KUKA KRL program: MyProgram_265().src

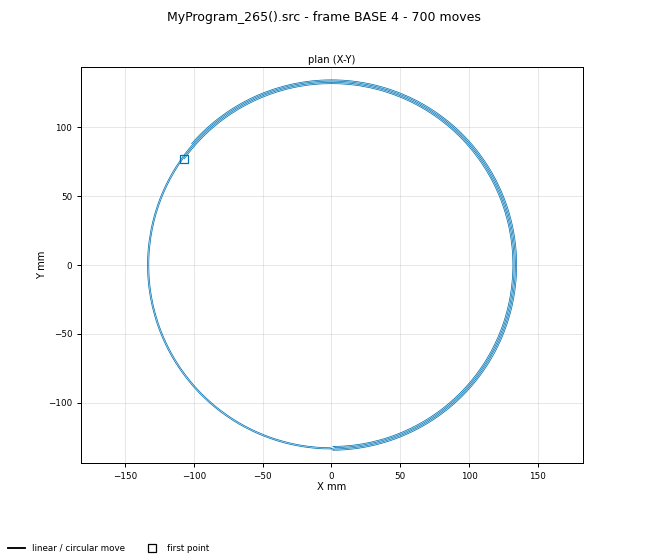
[picture p0: tool path of MyProgram_265().src in frame BASE 4, 700 of 700 moves have a stored position in this frame; points joined in program order, loops and branches not executed]
&ACCESS RVP
&REL 1
&PARAM TEMPLATE = C:\KRC\Roboter\Template\vorgabe
&PARAM EDITMASK = *
DEF MyProgram_265()
; ---- Setting reference (Base) ----
$BASE = BASE_DATA[4]

; --------------------------
; ---- Setting tool (TCP) ----
$TOOL = TOOL_DATA[3]
; --------------------------

$VEL.CP = VEL_APROX_PRINT
Startdeposition()
$VEL.CP = VEL_PRINT
LIN {X -106.8774,Y 77.2137,Z 169,A 144.3392,B 9.9671,C 0.0916,E1 9.8386,E2 306.7155} C_DIS
LIN {X -104.49,Y 80.4156,Z 169,A 142.5484,B 9.9671,C 0.0885,E1 9.8417,E2 308.5109} C_DIS
LIN {X -101.9162,Y 83.6531,Z 169,A 140.5928,B 9.9671,C 0.0871,E1 9.8451,E2 310.483} C_DIS
LIN {X -98.7876,Y 87.3252,Z 169,A 138.4779,B 9.9672,C 0.0828,E1 9.849,E2 312.5979} C_DIS
LIN {X -95.5133,Y 90.8953,Z 169,A 136.3519,B 9.9672,C 0.0786,E1 9.853,E2 314.724} C_DIS
LIN {X -92.6386,Y 93.824,Z 169,A 134.5368,B 9.9672,C 0.0754,E1 9.8566,E2 316.5411} C_DIS
LIN {X -89.1298,Y 97.1626,Z 169,A 132.4198,B 9.9672,C 0.0714,E1 9.8609,E2 318.6574} C_DIS
LIN {X -85.5317,Y 100.3446,Z 169,A 130.3464,B 9.9673,C 0.067,E1 9.8653,E2 320.7271} C_DIS
LIN {X -82.2873,Y 103.022,Z 169,A 128.4814,B 9.9673,C 0.0643,E1 9.8694,E2 322.5946} C_DIS
LIN {X -78.5317,Y 105.9128,Z 169,A 126.5407,B 9.9673,C 0.0584,E1 9.8736,E2 324.5197} C_DIS
LIN {X -75.9379,Y 107.7874,Z 169,A 125.1409,B 9.9673,C 0.0562,E1 9.8768,E2 325.9191} C_DIS
LIN {X -73.2593,Y 109.6255,Z 169,A 123.7103,B 9.9674,C 0.0542,E1 9.8801,E2 327.3506} C_DIS
LIN {X -70.5616,Y 111.3813,Z 169,A 122.3083,B 9.9674,C 0.052,E1 9.8834,E2 328.7518} C_DIS
LIN {X -67.8103,Y 113.0777,Z 169,A 120.8832,B 9.9674,C 0.0502,E1 9.8868,E2 330.1781} C_DIS
LIN {X -64.9859,Y 114.7243,Z 169,A 119.5244,B 9.9674,C 0.0469,E1 9.8901,E2 331.5284} C_DIS
LIN {X -62.1565,Y 116.2813,Z 169,A 118.0193,B 9.9674,C 0.0469,E1 9.8938,E2 333.0441} C_DIS
LIN {X -59.3244,Y 117.75,Z 169,A 116.6411,B 9.9674,C 0.0448,E1 9.8972,E2 334.4201} C_DIS
LIN {X -56.4217,Y 119.1678,Z 169,A 115.2277,B 9.9674,C 0.0431,E1 9.9008,E2 335.8334} C_DIS
LIN {X -53.4693,Y 120.5212,Z 169,A 113.8101,B 9.9674,C 0.0415,E1 9.9044,E2 337.2506} C_DIS
LIN {X -50.4743,Y 121.8058,Z 169,A 112.3819,B 9.9674,C 0.0401,E1 9.9081,E2 338.6791} C_DIS
LIN {X -47.4755,Y 123.0055,Z 169,A 110.9758,B 9.9674,C 0.0386,E1 9.9117,E2 340.0844} C_DIS
LIN {X -44.4123,Y 124.1444,Z 169,A 109.5673,B 9.9674,C 0.0369,E1 9.9154,E2 341.4904} C_DIS
LIN {X -41.359,Y 125.1947,Z 169,A 108.139,B 9.9674,C 0.036,E1 9.9192,E2 342.9206} C_DIS
LIN {X -38.2477,Y 126.1802,Z 169,A 106.716,B 9.9674,C 0.0348,E1 9.923,E2 344.3431} C_DIS
LIN {X -35.201,Y 127.0638,Z 169,A 105.3278,B 9.9674,C 0.0339,E1 9.9267,E2 345.7315} C_DIS
LIN {X -32.095,Y 127.8837,Z 169,A 103.9426,B 9.9674,C 0.0326,E1 9.9305,E2 347.1145} C_DIS
LIN {X -28.9319,Y 128.6366,Z 169,A 102.5542,B 9.9675,C 0.0311,E1 9.9342,E2 348.4991} C_DIS
LIN {X -25.7137,Y 129.3189,Z 169,A 101.0837,B 9.9675,C 0.0311,E1 9.9383,E2 349.9734} C_DIS
LIN {X -22.5381,Y 129.9106,Z 169,A 99.6804,B 9.9675,C 0.0303,E1 9.9421,E2 351.3759} C_DIS
LIN {X -19.3867,Y 130.4184,Z 169,A 98.2497,B 9.9675,C 0.0304,E1 9.9461,E2 352.8108} C_DIS
LIN {X -16.181,Y 130.854,Z 169,A 96.9617,B 9.9675,C 0.0275,E1 9.9496,E2 354.0843} C_DIS
LIN {X -12.9527,Y 131.2122,Z 169,A 95.4376,B 9.9675,C 0.0293,E1 9.9539,E2 355.6206} C_DIS
LIN {X -10.1839,Y 131.4569,Z 169,A 94.1244,B 9.9675,C 0.0311,E1 9.9576,E2 356.9454} C_DIS
LIN {X -6.5072,Y 131.6889,Z 169,A 92.6483,B 9.9675,C 0.0282,E1 9.9616,E2 358.4062} C_DIS
LIN {X -3.2367,Y 131.8105,Z 169,A 91.2707,B 9.9675,C 0.0272,E1 9.9655,E2 359.778} C_DIS
LIN {X -0.026,Y 131.8515,Z 169,A 89.7952,B 9.9675,C 0.0287,E1 9.9696,E2 361.2622} C_DIS
LIN {X 3.2431,Y 131.8103,Z 169,A 88.5531,B 9.9675,C 0.0251,E1 9.973,E2 362.4828} C_DIS
LIN {X 6.4726,Y 131.6906,Z 169,A 86.9955,B 9.9675,C 0.0283,E1 9.9774,E2 364.0576} C_DIS
LIN {X 9.6971,Y 131.4924,Z 169,A 85.5991,B 9.9675,C 0.0284,E1 9.9813,E2 365.4526} C_DIS
LIN {X 12.9671,Y 131.2108,Z 169,A 84.0255,B 9.9675,C 0.0318,E1 9.9857,E2 367.0428} C_DIS
LIN {X 17.2713,Y 130.7134,Z 169,A 82.2451,B 9.9675,C 0.0303,E1 9.9906,E2 368.8107} C_DIS
LIN {X 20.945,Y 130.1773,Z 169,A 80.6692,B 9.9675,C 0.0302,E1 9.995,E2 370.3819} C_DIS
LIN {X 24.0929,Y 129.6311,Z 169,A 79.2883,B 9.9675,C 0.0307,E1 9.9987,E2 371.7615} C_DIS
LIN {X 27.2612,Y 129.0015,Z 169,A 77.8766,B 9.9675,C 0.0316,E1 10.0026,E2 373.1737} C_DIS
LIN {X 30.4672,Y 128.2816,Z 169,A 76.4611,B 9.9675,C 0.0322,E1 10.0065,E2 374.5874} C_DIS
LIN {X 33.0736,Y 127.6354,Z 169,A 75.1852,B 9.9675,C 0.0353,E1 10.0099,E2 375.8757} C_DIS
LIN {X 36.7115,Y 126.6357,Z 169,A 73.6812,B 9.9675,C 0.0337,E1 10.0139,E2 377.3637} C_DIS
LIN {X 39.7849,Y 125.7039,Z 169,A 72.2874,B 9.9675,C 0.0348,E1 10.0177,E2 378.7571} C_DIS
LIN {X 42.8518,Y 124.6918,Z 169,A 70.9049,B 9.9675,C 0.0356,E1 10.0213,E2 380.1369} C_DIS
LIN {X 45.9047,Y 123.6004,Z 169,A 69.4777,B 9.9675,C 0.0374,E1 10.0251,E2 381.5662} C_DIS
LIN {X 48.9596,Y 122.4225,Z 169,A 68.0862,B 9.9675,C 0.0382,E1 10.0287,E2 382.9539} C_DIS
LIN {X 51.9473,Y 121.185,Z 169,A 66.679,B 9.9675,C 0.0398,E1 10.0323,E2 384.3612} C_DIS
LIN {X 54.905,Y 119.8742,Z 169,A 65.3074,B 9.9675,C 0.0407,E1 10.0358,E2 385.7289} C_DIS
LIN {X 57.3093,Y 118.7437,Z 169,A 64.0084,B 9.9675,C 0.0452,E1 10.0391,E2 387.0447} C_DIS
LIN {X 60.2841,Y 117.2615,Z 169,A 62.6301,B 9.9675,C 0.0456,E1 10.0425,E2 388.4154} C_DIS
LIN {X 63.5459,Y 115.5281,Z 169,A 61.1059,B 9.9675,C 0.046,E1 10.0462,E2 389.9303} C_DIS
LIN {X 66.3562,Y 113.9371,Z 169,A 59.7046,B 9.9675,C 0.048,E1 10.0496,E2 391.3314} C_DIS
LIN {X 69.1671,Y 112.2527,Z 169,A 58.2922,B 9.9675,C 0.0498,E1 10.053,E2 392.7426} C_DIS
LIN {X 71.9319,Y 110.5012,Z 169,A 56.8911,B 9.9675,C 0.0516,E1 10.0563,E2 394.1415} C_DIS
LIN {X 74.5745,Y 108.7351,Z 169,A 55.5407,B 9.9675,C 0.0531,E1 10.0594,E2 395.4885} C_DIS
LIN {X 77.241,Y 106.8575,Z 169,A 54.1443,B 9.9675,C 0.055,E1 10.0626,E2 396.8827} C_DIS
LIN {X 79.8287,Y 104.9389,Z 169,A 52.7306,B 9.9674,C 0.0577,E1 10.0657,E2 398.2984} C_DIS
LIN {X 82.4043,Y 102.9288,Z 169,A 51.1566,B 9.9674,C 0.0636,E1 10.0692,E2 399.8907} C_DIS
LIN {X 85.5078,Y 100.3649,Z 169,A 49.427,B 9.9674,C 0.0664,E1 10.0729,E2 401.6185} C_DIS
LIN {X 88.551,Y 97.6904,Z 169,A 47.6868,B 9.9674,C 0.0693,E1 10.0765,E2 403.3568} C_DIS
LIN {X 92.0675,Y 94.3843,Z 169,A 45.7593,B 9.9674,C 0.0697,E1 10.0804,E2 405.2652} C_DIS
LIN {X 94.9298,Y 91.5046,Z 169,A 43.8603,B 9.9673,C 0.0763,E1 10.0841,E2 407.1806} C_DIS
LIN {X 97.7032,Y 88.5369,Z 169,A 42.1172,B 9.9673,C 0.0796,E1 10.0874,E2 408.9218} C_DIS
LIN {X 100.3808,Y 85.4891,Z 169,A 40.3789,B 9.9673,C 0.0828,E1 10.0906,E2 410.658} C_DIS
LIN {X 102.9666,Y 82.3569,Z 169,A 38.639,B 9.9672,C 0.0862,E1 10.0936,E2 412.3958} C_DIS
LIN {X 105.8792,Y 78.5769,Z 169,A 36.7305,B 9.9672,C 0.0872,E1 10.0968,E2 414.2859} C_DIS
LIN {X 107.3485,Y 76.5572,Z 169,A 35.5161,B 9.9672,C 0.0927,E1 10.0988,E2 415.516} C_DIS
LIN {X 109.6294,Y 73.2536,Z 169,A 33.9386,B 9.9672,C 0.093,E1 10.1013,E2 417.0748} C_DIS
LIN {X 111.3712,Y 70.5777,Z 169,A 32.5709,B 9.9671,C 0.0959,E1 10.1033,E2 418.441} C_DIS
LIN {X 113.0732,Y 67.8178,Z 169,A 31.1149,B 9.9671,C 0.1005,E1 10.1055,E2 419.9033} C_DIS
LIN {X 114.7841,Y 64.8799,Z 169,A 29.7352,B 9.9671,C 0.1019,E1 10.1074,E2 421.2725} C_DIS
LIN {X 116.2924,Y 62.1357,Z 169,A 28.3549,B 9.967,C 0.1058,E1 10.1092,E2 422.6559} C_DIS
LIN {X 117.7557,Y 59.3133,Z 169,A 27.0047,B 9.967,C 0.1087,E1 10.1109,E2 424.0033} C_DIS
LIN {X 119.1743,Y 56.4081,Z 169,A 25.62,B 9.967,C 0.1118,E1 10.1126,E2 425.3865} C_DIS
LIN {X 120.5203,Y 53.4713,Z 169,A 24.2359,B 9.9669,C 0.1151,E1 10.1142,E2 426.7693} C_DIS
LIN {X 121.7955,Y 50.499,Z 169,A 22.8442,B 9.9669,C 0.1185,E1 10.1157,E2 428.1603} C_DIS
LIN {X 123.0031,Y 47.4818,Z 169,A 21.4588,B 9.9669,C 0.1217,E1 10.1171,E2 429.5436} C_DIS
LIN {X 124.1429,Y 44.4166,Z 169,A 20.0581,B 9.9668,C 0.1251,E1 10.1184,E2 430.9429} C_DIS
LIN {X 125.0907,Y 41.6715,Z 169,A 18.7574,B 9.9668,C 0.1294,E1 10.1196,E2 432.2491} C_DIS
LIN {X 126.1752,Y 38.2641,Z 169,A 17.2961,B 9.9667,C 0.1316,E1 10.1208,E2 433.7007} C_DIS
LIN {X 127.0596,Y 35.2158,Z 169,A 16.006,B 9.9667,C 0.1333,E1 10.1218,E2 434.9813} C_DIS
LIN {X 127.8876,Y 32.0798,Z 169,A 14.5795,B 9.9667,C 0.1377,E1 10.1228,E2 436.4111} C_DIS
LIN {X 128.5443,Y 29.3357,Z 169,A 13.2661,B 9.9665,C 0.1432,E1 10.1236,E2 437.7358} C_DIS
LIN {X 129.3167,Y 25.7247,Z 169,A 11.7507,B 9.9665,C 0.1457,E1 10.1245,E2 439.242} C_DIS
LIN {X 129.9091,Y 22.5464,Z 169,A 10.3707,B 9.9665,C 0.1491,E1 10.1252,E2 440.6204} C_DIS
LIN {X 130.4172,Y 19.395,Z 169,A 8.9639,B 9.9664,C 0.1536,E1 10.1258,E2 442.0308} C_DIS
LIN {X 130.8537,Y 16.1835,Z 169,A 7.6069,B 9.9664,C 0.1564,E1 10.1263,E2 443.3828} C_DIS
LIN {X 131.2111,Y 12.9638,Z 169,A 6.1987,B 9.9663,C 0.1605,E1 10.1267,E2 444.7924} C_DIS
LIN {X 131.4627,Y 10.1046,Z 169,A 4.8935,B 9.9662,C 0.1655,E1 10.127,E2 446.1056} C_DIS
LIN {X 131.6884,Y 6.5173,Z 169,A 3.4541,B 9.9662,C 0.1671,E1 10.1272,E2 447.5319} C_DIS
LIN {X 131.8107,Y 3.2292,Z 169,A 2.061,B 9.9662,C 0.1704,E1 10.1273,E2 448.9221} C_DIS
LIN {X 131.8522,Y 0.2318,Z 169,A 0.6856,B 9.966,C 0.176,E1 10.1273,E2 450.3075} C_DIS
LIN {X 131.8106,Y -3.2343,Z 169,A -0.7295,B 9.966,C 0.1782,E1 10.1273,E2 451.713} C_DIS
LIN {X 131.691,Y -6.4646,Z 169,A -2.015,B 9.966,C 0.1795,E1 10.1271,E2 452.9857} C_DIS
LIN {X 131.4921,Y -9.7022,Z 169,A -3.4963,B 9.9658,C 0.1853,E1 10.1269,E2 454.477} C_DIS
LIN {X 131.2186,Y -12.8854,Z 169,A -4.8644,B 9.9658,C 0.1889,E1 10.1265,E2 455.8441} C_DIS
LIN {X 130.859,Y -16.1387,Z 169,A -6.2578,B 9.9658,C 0.1923,E1 10.1261,E2 457.2355} C_DIS
LIN {X 130.431,Y -19.2984,Z 169,A -7.6232,B 9.9656,C 0.1959,E1 10.1255,E2 458.6} C_DIS
LIN {X 129.9116,Y -22.5325,Z 169,A -8.9978,B 9.9656,C 0.1988,E1 10.1249,E2 459.9701} C_DIS
LIN {X 129.326,Y -25.6791,Z 169,A -10.4159,B 9.9655,C 0.2035,E1 10.1242,E2 461.393} C_DIS
LIN {X 128.6466,Y -28.888,Z 169,A -11.816,B 9.9655,C 0.207,E1 10.1233,E2 462.7915} C_DIS
LIN {X 127.8992,Y -32.0341,Z 169,A -13.2076,B 9.9653,C 0.2107,E1 10.1224,E2 464.183} C_DIS
LIN {X 127.0798,Y -35.1435,Z 169,A -14.5851,B 9.9653,C 0.2142,E1 10.1214,E2 465.5596} C_DIS
LIN {X 126.1828,Y -38.2391,Z 169,A -16.0454,B 9.9652,C 0.2195,E1 10.1202,E2 467.0286} C_DIS
LIN {X 124.9065,Y -42.2245,Z 169,A -17.8958,B 9.965,C 0.2254,E1 10.1186,E2 468.8848} C_DIS
LIN {X 123.6012,Y -45.9026,Z 169,A -19.4299,B 9.965,C 0.2263,E1 10.1172,E2 470.4013} C_DIS
LIN {X 122.4235,Y -48.9571,Z 169,A -20.8082,B 9.965,C 0.2292,E1 10.1158,E2 471.7758} C_DIS
LIN {X 121.1855,Y -51.9463,Z 169,A -22.2141,B 9.9649,C 0.233,E1 10.1142,E2 473.1832} C_DIS
LIN {X 119.8648,Y -54.9253,Z 169,A -23.5996,B 9.9648,C 0.2361,E1 10.1127,E2 474.5666} C_DIS
LIN {X 118.4854,Y -57.8418,Z 169,A -24.9809,B 9.9648,C 0.2394,E1 10.111,E2 475.9469} C_DIS
LIN {X 117.0349,Y -60.7239,Z 169,A -26.3094,B 9.9647,C 0.2414,E1 10.1093,E2 477.2681} C_DIS
LIN {X 115.5353,Y -63.5329,Z 169,A -27.7352,B 9.9645,C 0.246,E1 10.1074,E2 478.7005} C_DIS
LIN {X 113.9475,Y -66.3382,Z 169,A -29.1224,B 9.9645,C 0.2493,E1 10.1055,E2 480.0876} C_DIS
LIN {X 112.2709,Y -69.1374,Z 169,A -30.5256,B 9.9644,C 0.2525,E1 10.1034,E2 481.4906} C_DIS
LIN {X 110.2507,Y -72.3153,Z 169,A -32.2569,B 9.9642,C 0.2589,E1 10.1008,E2 483.2351} C_DIS
LIN {X 107.7951,Y -75.927,Z 169,A -34.0046,B 9.9642,C 0.26,E1 10.0981,E2 484.9667} C_DIS
LIN {X 105.9051,Y -78.5421,Z 169,A -35.386,B 9.9642,C 0.263,E1 10.0958,E2 486.3471} C_DIS
LIN {X 104.4254,Y -80.4992,Z 169,A -36.5931,B 9.964,C 0.2688,E1 10.0937,E2 487.5724} C_DIS
LIN {X 101.8901,Y -83.6851,Z 169,A -38.3507,B 9.9639,C 0.2726,E1 10.0906,E2 489.3304} C_DIS
LIN {X 98.7684,Y -87.3469,Z 169,A -40.4118,B 9.9637,C 0.2767,E1 10.0868,E2 491.3901} C_DIS
LIN {X 95.5049,Y -90.9041,Z 169,A -42.4828,B 9.9637,C 0.2807,E1 10.0829,E2 493.4601} C_DIS
LIN {X 92.6078,Y -93.8543,Z 169,A -44.2682,B 9.9635,C 0.2843,E1 10.0794,E2 495.246} C_DIS
LIN {X 89.1247,Y -97.1673,Z 169,A -46.3322,B 9.9635,C 0.2881,E1 10.0752,E2 497.309} C_DIS
LIN {X 85.5204,Y -100.3542,Z 169,A -48.3987,B 9.9633,C 0.2917,E1 10.0708,E2 499.3747} C_DIS
LIN {X 82.358,Y -102.9657,Z 169,A -50.1566,B 9.9633,C 0.2946,E1 10.067,E2 501.1314} C_DIS
LIN {X 78.5751,Y -105.8805,Z 169,A -52.0711,B 9.9633,C 0.2948,E1 10.0628,E2 503.0285} C_DIS
LIN {X 75.9621,Y -107.7703,Z 169,A -53.4748,B 9.9632,C 0.2974,E1 10.0596,E2 504.4338} C_DIS
LIN {X 72.5727,Y -110.0813,Z 169,A -55.2404,B 9.9631,C 0.3001,E1 10.0555,E2 506.199} C_DIS
LIN {X 69.1643,Y -112.2544,Z 169,A -56.9607,B 9.9631,C 0.3022,E1 10.0514,E2 507.9167} C_DIS
LIN {X 66.3665,Y -113.9311,Z 169,A -58.3647,B 9.963,C 0.3041,E1 10.0481,E2 509.3203} C_DIS
LIN {X 63.5661,Y -115.5169,Z 169,A -59.7625,B 9.9629,C 0.3062,E1 10.0446,E2 510.7193} C_DIS
LIN {X 60.7608,Y -117.0155,Z 169,A -61.1372,B 9.9629,C 0.3081,E1 10.0412,E2 512.0942} C_DIS
LIN {X 57.8826,Y -118.4652,Z 169,A -62.5279,B 9.9628,C 0.3099,E1 10.0378,E2 513.485} C_DIS
LIN {X 54.9401,Y -119.858,Z 169,A -63.9294,B 9.9628,C 0.3115,E1 10.0342,E2 514.8861} C_DIS
LIN {X 51.9832,Y -121.1695,Z 169,A -65.3247,B 9.9627,C 0.313,E1 10.0306,E2 516.2812} C_DIS
LIN {X 48.8175,Y -122.4797,Z 169,A -66.7966,B 9.9627,C 0.3145,E1 10.0268,E2 517.7524} C_DIS
LIN {X 45.9072,Y -123.5995,Z 169,A -68.1518,B 9.9626,C 0.316,E1 10.0233,E2 519.1086} C_DIS
LIN {X 42.8223,Y -124.702,Z 169,A -69.7168,B 9.9624,C 0.3207,E1 10.0191,E2 520.6918} C_DIS
LIN {X 38.8604,Y -125.9927,Z 169,A -71.4795,B 9.9624,C 0.3214,E1 10.0144,E2 522.4501} C_DIS
LIN {X 35.2363,Y -127.0539,Z 169,A -73.0067,B 9.9624,C 0.3205,E1 10.0104,E2 523.9646} C_DIS
LIN {X 32.0725,Y -127.8894,Z 169,A -74.412,B 9.9624,C 0.3213,E1 10.0066,E2 525.369} C_DIS
LIN {X 28.9296,Y -128.6371,Z 169,A -75.8087,B 9.9624,C 0.3223,E1 10.0028,E2 526.7658} C_DIS
LIN {X 25.7271,Y -129.3162,Z 169,A -77.2229,B 9.9624,C 0.3231,E1 9.9989,E2 528.18} C_DIS
LIN {X 22.5399,Y -129.9103,Z 169,A -78.6228,B 9.9624,C 0.3238,E1 9.9951,E2 529.5796} C_DIS
LIN {X 19.3793,Y -130.4195,Z 169,A -80.0488,B 9.9623,C 0.3254,E1 9.9911,E2 531.0108} C_DIS
LIN {X 16.1804,Y -130.854,Z 169,A -81.434,B 9.9623,C 0.3257,E1 9.9873,E2 532.3946} C_DIS
LIN {X 12.9655,Y -131.2109,Z 169,A -82.8418,B 9.9623,C 0.3263,E1 9.9834,E2 533.8035} C_DIS
LIN {X 9.7296,Y -131.4901,Z 169,A -84.235,B 9.9623,C 0.3264,E1 9.9795,E2 535.1952} C_DIS
LIN {X 6.5046,Y -131.689,Z 169,A -85.6292,B 9.9623,C 0.3266,E1 9.9756,E2 536.589} C_DIS
LIN {X 3.2349,Y -131.8106,Z 169,A -87.0343,B 9.9623,C 0.3266,E1 9.9717,E2 537.9928} C_DIS
LIN {X 0.956,Y -131.8451,Z 169,A -87.7495,B 9.9624,C 0.321,E1 9.9698,E2 538.6752} C_DIS
Enddeposition()
LIN {X 0.956,Y -131.8451,Z 169,A -87.7495,B 9.9624,C 0.321,E1 9.9698,E2 538.6752} C_DIS
Startdeposition()
$VEL.CP = VEL_PRINT
LIN {X 3.133,Y -132.7261,Z 169,A -86.3062,B 9.9633,C 0.3159,E1 9.9747,E2 537.2036} C_DIS
LIN {X 6.6755,Y -132.5939,Z 169,A -84.9357,B 9.9633,C 0.319,E1 9.9784,E2 535.852} C_DIS
LIN {X 10.3215,Y -132.3616,Z 169,A -83.3705,B 9.9633,C 0.3187,E1 9.9828,E2 534.2874} C_DIS
LIN {X 13.2936,Y -132.096,Z 169,A -81.9074,B 9.9633,C 0.3144,E1 9.9869,E2 532.802} C_DIS
LIN {X 17.2969,Y -131.6302,Z 169,A -80.3789,B 9.9633,C 0.3181,E1 9.9911,E2 531.2983} C_DIS
LIN {X 20.4371,Y -131.1793,Z 169,A -78.9281,B 9.9633,C 0.3156,E1 9.9951,E2 529.8366} C_DIS
LIN {X 24.5903,Y -130.4649,Z 169,A -77.0814,B 9.9634,C 0.3138,E1 10.0002,E2 527.9854} C_DIS
LIN {X 27.6052,Y -129.8606,Z 169,A -75.7814,B 9.9634,C 0.3134,E1 10.0037,E2 526.6878} C_DIS
LIN {X 30.6136,Y -129.1848,Z 169,A -74.6207,B 9.9634,C 0.3162,E1 10.0068,E2 525.5472} C_DIS
LIN {X 33.4173,Y -128.4894,Z 169,A -73.2702,B 9.9634,C 0.3128,E1 10.0105,E2 524.183} C_DIS
LIN {X 39.0819,Y -126.879,Z 169,A -70.7402,B 9.9635,C 0.3107,E1 10.0173,E2 521.6525} C_DIS
LIN {X 44.8545,Y -124.9548,Z 169,A -68.0494,B 9.9636,C 0.3065,E1 10.0245,E2 518.9518} C_DIS
LIN {X 50.4355,Y -122.8107,Z 169,A -65.5025,B 9.9637,C 0.3042,E1 10.0311,E2 516.4071} C_DIS
LIN {X 53.6522,Y -121.4388,Z 169,A -64.1366,B 9.9637,C 0.3055,E1 10.0345,E2 515.0575} C_DIS
LIN {X 57.0509,Y -119.8783,Z 169,A -62.0622,B 9.964,C 0.2928,E1 10.0399,E2 512.9248} C_DIS
LIN {X 60.3518,Y -118.2508,Z 169,A -60.9337,B 9.9638,C 0.3011,E1 10.0426,E2 511.8518} C_DIS
LIN {X 63.3275,Y -116.6868,Z 169,A -59.3333,B 9.964,C 0.2955,E1 10.0466,E2 510.2319} C_DIS
LIN {X 66.8934,Y -114.6801,Z 169,A -57.2048,B 9.9643,C 0.2844,E1 10.0519,E2 508.0568} C_DIS
LIN {X 70.4447,Y -112.5334,Z 169,A -55.7813,B 9.9641,C 0.29,E1 10.0551,E2 506.6771} C_DIS
LIN {X 74.0878,Y -110.1693,Z 169,A -54.1118,B 9.9641,C 0.2915,E1 10.059,E2 505.0312} C_DIS
LIN {X 76.9831,Y -108.1656,Z 169,A -52.5715,B 9.9641,C 0.2883,E1 10.0625,E2 503.4869} C_DIS
LIN {X 80.0917,Y -105.8841,Z 169,A -50.8654,B 9.9643,C 0.2843,E1 10.0663,E2 501.774} C_DIS
LIN {X 83.688,Y -103.066,Z 169,A -48.8178,B 9.9644,C 0.2787,E1 10.0708,E2 499.7151} C_DIS
LIN {X 86.8545,Y -100.4116,Z 169,A -47.3308,B 9.9644,C 0.2821,E1 10.0739,E2 498.2629} C_DIS
LIN {X 89.3604,Y -98.1879,Z 169,A -44.8651,B 9.9651,C 0.2551,E1 10.0793,E2 495.6693} C_DIS
LIN {X 93.9167,Y -93.8398,Z 169,A -42.9682,B 9.9647,C 0.2688,E1 10.0828,E2 493.8717} C_DIS
LIN {X 96.7874,Y -90.8757,Z 169,A -41.0498,B 9.9649,C 0.2616,E1 10.0866,E2 491.9345} C_DIS
LIN {X 99.0609,Y -88.3918,Z 169,A -39.1472,B 9.9653,C 0.2477,E1 10.0902,E2 489.9745} C_DIS
LIN {X 102.5783,Y -84.2847,Z 169,A -37.4277,B 9.965,C 0.2569,E1 10.0931,E2 488.3288} C_DIS
LIN {X 104.9344,Y -81.3319,Z 169,A -35.8765,B 9.965,C 0.2549,E1 10.0958,E2 486.7856} C_DIS
LIN {X 107.3946,Y -78.0546,Z 169,A -34.0786,B 9.9652,C 0.25,E1 10.0988,E2 484.9821} C_DIS
LIN {X 110.1674,Y -74.0905,Z 169,A -31.9876,B 9.9653,C 0.2447,E1 10.1021,E2 482.8885} C_DIS
LIN {X 112.5414,Y -70.432,Z 169,A -30.3096,B 9.9653,C 0.2449,E1 10.1046,E2 481.2336} C_DIS
LIN {X 115.1575,Y -66.0679,Z 169,A -28.102,B 9.9655,C 0.239,E1 10.1077,E2 479.0222} C_DIS
LIN {X 116.8558,Y -63.0148,Z 169,A -26.535,B 9.9655,C 0.2336,E1 10.1098,E2 477.4463} C_DIS
LIN {X 118.5812,Y -59.7027,Z 169,A -25.0195,B 9.9656,C 0.2316,E1 10.1117,E2 475.9408} C_DIS
LIN {X 120.046,Y -56.6999,Z 169,A -23.1071,B 9.966,C 0.2164,E1 10.1141,E2 473.9688} C_DIS
LIN {X 121.7842,Y -52.8605,Z 169,A -21.7558,B 9.9658,C 0.2228,E1 10.1156,E2 472.6732} C_DIS
LIN {X 123.6907,Y -48.2309,Z 169,A -19.7016,B 9.9659,C 0.2194,E1 10.1177,E2 470.6297} C_DIS
LIN {X 124.6995,Y -45.5627,Z 169,A -18.5054,B 9.9659,C 0.2168,E1 10.1188,E2 469.4365} C_DIS
LIN {X 126.3315,Y -40.8187,Z 169,A -16.2885,B 9.9661,C 0.2095,E1 10.1208,E2 467.211} C_DIS
LIN {X 127.5706,Y -36.7651,Z 169,A -14.0529,B 9.9664,C 0.1945,E1 10.1226,E2 464.9234} C_DIS
LIN {X 128.6447,Y -32.8056,Z 169,A -13.0042,B 9.9662,C 0.207,E1 10.1233,E2 463.9614} C_DIS
LIN {X 129.315,Y -30.0586,Z 169,A -11.4905,B 9.9664,C 0.1964,E1 10.1243,E2 462.4106} C_DIS
LIN {X 129.9474,Y -27.2009,Z 169,A -10.2533,B 9.9664,C 0.1934,E1 10.125,E2 461.1753} C_DIS
LIN {X 130.6623,Y -23.5171,Z 169,A -8.8165,B 9.9664,C 0.1931,E1 10.1258,E2 459.7591} C_DIS
LIN {X 131.2763,Y -19.8106,Z 169,A -6.9997,B 9.9666,C 0.1837,E1 10.1266,E2 457.9168} C_DIS
LIN {X 131.7838,Y -16.089,Z 169,A -5.5433,B 9.9666,C 0.183,E1 10.1271,E2 456.4788} C_DIS
LIN {X 132.0968,Y -13.2852,Z 169,A -4.315,B 9.9667,C 0.1792,E1 10.1274,E2 455.2481} C_DIS
LIN {X 132.3693,Y -10.2168,Z 169,A -2.9587,B 9.9667,C 0.1746,E1 10.1277,E2 453.887} C_DIS
LIN {X 132.5908,Y -6.739,Z 169,A -1.5134,B 9.9668,C 0.1716,E1 10.128,E2 452.4474} C_DIS
LIN {X 132.7285,Y -3.0465,Z 169,A 0.0159,B 9.9668,C 0.1686,E1 10.128,E2 450.9245} C_DIS
LIN {X 132.7651,Y -0.1633,Z 169,A 1.2664,B 9.967,C 0.1648,E1 10.1281,E2 449.6721} C_DIS
LIN {X 132.7048,Y 3.9009,Z 169,A 3.0209,B 9.967,C 0.1597,E1 10.128,E2 447.9158} C_DIS
LIN {X 132.5403,Y 7.6815,Z 169,A 4.6581,B 9.9671,C 0.1548,E1 10.1278,E2 446.2765} C_DIS
LIN {X 132.2754,Y 11.3553,Z 169,A 6.1447,B 9.9671,C 0.1527,E1 10.1274,E2 444.801} C_DIS
LIN {X 131.8634,Y 15.4216,Z 169,A 7.9332,B 9.9672,C 0.147,E1 10.1269,E2 443.0079} C_DIS
LIN {X 131.3907,Y 19.0325,Z 169,A 9.4014,B 9.9672,C 0.1449,E1 10.1263,E2 441.5508} C_DIS
LIN {X 130.9277,Y 21.9914,Z 169,A 10.7864,B 9.9673,C 0.139,E1 10.1257,E2 440.1534} C_DIS
LIN {X 130.157,Y 26.1705,Z 169,A 12.3166,B 9.9673,C 0.1411,E1 10.1249,E2 438.6585} C_DIS
LIN {X 129.5089,Y 29.2098,Z 169,A 13.8793,B 9.9674,C 0.1319,E1 10.124,E2 437.0678} C_DIS
LIN {X 128.7008,Y 32.5846,Z 169,A 15.3067,B 9.9674,C 0.1294,E1 10.123,E2 435.6477} C_DIS
LIN {X 127.461,Y 37.1394,Z 169,A 18.0423,B 9.9677,C 0.1069,E1 10.1209,E2 432.8252} C_DIS
LIN {X 125.8145,Y 42.3856,Z 169,A 19.7214,B 9.9677,C 0.1171,E1 10.1195,E2 431.229} C_DIS
LIN {X 124.7232,Y 45.4969,Z 169,A 21.1767,B 9.9677,C 0.1124,E1 10.1181,E2 429.7687} C_DIS
LIN {X 123.5178,Y 48.6758,Z 169,A 22.637,B 9.9677,C 0.1086,E1 10.1166,E2 428.3081} C_DIS
LIN {X 121.8728,Y 52.6556,Z 169,A 24.3208,B 9.9677,C 0.1078,E1 10.1148,E2 426.6441} C_DIS
LIN {X 120.5497,Y 55.618,Z 169,A 25.5166,B 9.9677,C 0.109,E1 10.1134,E2 425.472} C_DIS
LIN {X 119.3338,Y 58.1842,Z 169,A 27.0277,B 9.9678,C 0.099,E1 10.1116,E2 423.9257} C_DIS
LIN {X 117.6252,Y 61.5622,Z 169,A 28.4118,B 9.9678,C 0.1007,E1 10.1098,E2 422.5706} C_DIS
LIN {X 113.9997,Y 68.0455,Z 169,A 31.7897,B 9.9679,C 0.0887,E1 10.1052,E2 419.1702} C_DIS
LIN {X 111.8821,Y 71.4739,Z 169,A 33.3838,B 9.9679,C 0.0878,E1 10.1028,E2 417.5926} C_DIS
LIN {X 109.7665,Y 74.6828,Z 169,A 35.0615,B 9.9679,C 0.0834,E1 10.1002,E2 415.9117} C_DIS
LIN {X 107.2675,Y 78.23,Z 169,A 37.0641,B 9.968,C 0.076,E1 10.0969,E2 413.8924} C_DIS
LIN {X 104.5054,Y 81.8826,Z 169,A 39.3061,B 9.968,C 0.0653,E1 10.093,E2 411.6173} C_DIS
LIN {X 102.0128,Y 84.9685,Z 169,A 40.6918,B 9.968,C 0.0691,E1 10.0906,E2 410.2704} C_DIS
LIN {X 99.0595,Y 88.3934,Z 169,A 42.6057,B 9.968,C 0.0658,E1 10.0871,E2 408.3601} C_DIS
LIN {X 96.2514,Y 91.4435,Z 169,A 44.3927,B 9.9681,C 0.0621,E1 10.0837,E2 406.5727} C_DIS
LIN {X 93.326,Y 94.4272,Z 169,A 46.1406,B 9.9681,C 0.0597,E1 10.0803,E2 404.8308} C_DIS
LIN {X 90.3234,Y 97.3028,Z 169,A 47.8988,B 9.9681,C 0.057,E1 10.0767,E2 403.0763} C_DIS
LIN {X 87.023,Y 100.2658,Z 169,A 49.8319,B 9.9681,C 0.0529,E1 10.0726,E2 401.1405} C_DIS
LIN {X 83.6609,Y 103.0879,Z 169,A 51.6018,B 9.9681,C 0.0523,E1 10.0689,E2 399.385} C_DIS
LIN {X 79.8914,Y 106.0352,Z 169,A 53.7379,B 9.9681,C 0.0471,E1 10.0641,E2 397.2399} C_DIS
LIN {X 76.4169,Y 108.566,Z 169,A 55.3668,B 9.9681,C 0.0491,E1 10.0605,E2 395.6376} C_DIS
LIN {X 71.6665,Y 111.7588,Z 169,A 58.0234,B 9.9682,C 0.041,E1 10.0543,E2 392.9585} C_DIS
LIN {X 68.5445,Y 113.7004,Z 169,A 59.6056,B 9.9682,C 0.0388,E1 10.0505,E2 391.3767} C_DIS
LIN {X 65.608,Y 115.4198,Z 169,A 60.8851,B 9.9682,C 0.0409,E1 10.0474,E2 390.1195} C_DIS
LIN {X 63.4738,Y 116.6071,Z 169,A 62.0825,B 9.9682,C 0.0362,E1 10.0445,E2 388.9049} C_DIS
LIN {X 60.5076,Y 118.1715,Z 169,A 63.4866,B 9.9682,C 0.0353,E1 10.041,E2 387.5059} C_DIS
LIN {X 55.2198,Y 120.7338,Z 169,A 65.993,B 9.9682,C 0.0329,E1 10.0347,E2 385.0031} C_DIS
LIN {X 51.2689,Y 122.4626,Z 169,A 67.7954,B 9.9682,C 0.0321,E1 10.0301,E2 383.2077} C_DIS
LIN {X 48.5583,Y 123.5634,Z 169,A 69.1399,B 9.9682,C 0.029,E1 10.0266,E2 381.8536} C_DIS
LIN {X 45.8202,Y 124.6063,Z 169,A 70.4525,B 9.9682,C 0.0267,E1 10.0231,E2 380.5354} C_DIS
LIN {X 42.8534,Y 125.6569,Z 169,A 71.8376,B 9.9682,C 0.0249,E1 10.0195,E2 379.1473} C_DIS
LIN {X 39.6165,Y 126.7154,Z 169,A 73.1404,B 9.9682,C 0.0272,E1 10.016,E2 377.8646} C_DIS
LIN {X 35.2587,Y 127.995,Z 169,A 75.5171,B 9.9682,C 0.0168,E1 10.0095,E2 375.4386} C_DIS
LIN {X 31.5801,Y 128.9518,Z 169,A 76.8053,B 9.9682,C 0.0232,E1 10.0061,E2 374.1928} C_DIS
LIN {X 28.3176,Y 129.7068,Z 169,A 78.219,B 9.9682,C 0.023,E1 10.0023,E2 372.7831} C_DIS
LIN {X 24.1033,Y 130.5573,Z 169,A 80.0778,B 9.9682,C 0.022,E1 9.9972,E2 370.9245} C_DIS
LIN {X 21.0109,Y 131.0905,Z 169,A 81.3654,B 9.9682,C 0.0228,E1 9.9937,E2 369.6452} C_DIS
LIN {X 17.8564,Y 131.5568,Z 169,A 82.8129,B 9.9682,C 0.0208,E1 9.9896,E2 368.1897} C_DIS
LIN {X 14.8754,Y 131.9275,Z 169,A 84.132,B 9.9682,C 0.02,E1 9.986,E2 366.8683} C_DIS
LIN {X 11.0545,Y 132.3008,Z 169,A 85.7001,B 9.9682,C 0.0214,E1 9.9817,E2 365.3113} C_DIS
LIN {X 7.0357,Y 132.5758,Z 169,A 87.4941,B 9.9682,C 0.02,E1 9.9766,E2 363.5114} C_DIS
LIN {X 3.4007,Y 132.7187,Z 169,A 89.0046,B 9.9682,C 0.0211,E1 9.9724,E2 362.0086} C_DIS
LIN {X -0.378,Y 132.7619,Z 169,A 90.7141,B 9.9682,C 0.0196,E1 9.9676,E2 360.2905} C_DIS
LIN {X -4.3263,Y 132.6929,Z 169,A 92.3876,B 9.9682,C 0.0204,E1 9.963,E2 358.6215} C_DIS
LIN {X -7.4689,Y 132.5534,Z 169,A 93.7465,B 9.9682,C 0.0206,E1 9.9592,E2 357.2632} C_DIS
LIN {X -10.4719,Y 132.3501,Z 169,A 95.1888,B 9.9682,C 0.018,E1 9.9551,E2 355.8046} C_DIS
LIN {X -14.9687,Y 131.9174,Z 169,A 96.9345,B 9.9682,C 0.0228,E1 9.9504,E2 354.0842} C_DIS
LIN {X -18.1316,Y 131.5194,Z 169,A 98.2722,B 9.9682,C 0.0242,E1 9.9467,E2 352.7518} C_DIS
LIN {X -21.96,Y 130.9329,Z 169,A 100.0924,B 9.9682,C 0.022,E1 9.9416,E2 350.915} C_DIS
LIN {X -26.3582,Y 130.1188,Z 169,A 101.9881,B 9.9682,C 0.0238,E1 9.9364,E2 349.0245} C_DIS
LIN {X -29.6878,Y 129.3998,Z 169,A 103.3351,B 9.9682,C 0.0272,E1 9.9328,E2 347.6931} C_DIS
LIN {X -34.854,Y 128.1065,Z 169,A 105.5071,B 9.9682,C 0.0315,E1 9.927,E2 345.5376} C_DIS
LIN {X -40.6753,Y 126.3773,Z 169,A 108.4316,B 9.9682,C 0.0279,E1 9.9191,E2 342.5793} C_DIS
LIN {X -45.179,Y 124.8378,Z 169,A 110.5261,B 9.9682,C 0.0291,E1 9.9135,E2 340.4816} C_DIS
LIN {X -48.2211,Y 123.6945,Z 169,A 112.1804,B 9.9682,C 0.0258,E1 9.9091,E2 338.7985} C_DIS
LIN {X -51.382,Y 122.4154,Z 169,A 113.2871,B 9.9682,C 0.0345,E1 9.9064,E2 337.7362} C_DIS
LIN {X -55.0283,Y 120.8224,Z 169,A 115.0256,B 9.9682,C 0.0362,E1 9.902,E2 335.9968} C_DIS
LIN {X -58.5567,Y 119.15,Z 169,A 116.5905,B 9.9682,C 0.0407,E1 9.8981,E2 334.4473} C_DIS
LIN {X -60.7074,Y 118.0698,Z 169,A 117.9228,B 9.9682,C 0.0365,E1 9.8947,E2 333.0813} C_DIS
LIN {X -64.2557,Y 116.1779,Z 169,A 119.6182,B 9.9682,C 0.0398,E1 9.8905,E2 331.3921} C_DIS
LIN {X -67.1727,Y 114.5161,Z 169,A 120.9029,B 9.9682,C 0.0451,E1 9.8875,E2 330.1282} C_DIS
LIN {X -69.5404,Y 113.094,Z 169,A 122.2331,B 9.9682,C 0.0443,E1 9.8842,E2 328.7826} C_DIS
LIN {X -71.7933,Y 111.6776,Z 169,A 123.7075,B 9.9682,C 0.04,E1 9.8807,E2 327.2707} C_DIS
LIN {X -74.8962,Y 109.6209,Z 169,A 125.9757,B 9.9682,C 0.0301,E1 9.8753,E2 324.9247} C_DIS
LIN {X -80.3861,Y 105.6612,Z 169,A 128.3925,B 9.9682,C 0.0449,E1 9.8701,E2 322.5712} C_DIS
LIN {X -83.5458,Y 103.1808,Z 169,A 129.7748,B 9.9682,C 0.0547,E1 9.8671,E2 321.2325} C_DIS
LIN {X -86.0558,Y 101.0965,Z 169,A 131.1832,B 9.9682,C 0.0574,E1 9.8641,E2 319.8254} C_DIS
LIN {X -89.4498,Y 98.1068,Z 169,A 133.1033,B 9.9682,C 0.0619,E1 9.8602,E2 317.9111} C_DIS
LIN {X -92.1199,Y 95.604,Z 169,A 134.8075,B 9.9682,C 0.0628,E1 9.8567,E2 316.1936} C_DIS
LIN {X -95.1581,Y 92.5805,Z 169,A 136.4781,B 9.9681,C 0.07,E1 9.8534,E2 314.5461} C_DIS
LIN {X -97.367,Y 90.2545,Z 169,A 137.9758,B 9.9681,C 0.0709,E1 9.8506,E2 313.0364} C_DIS
LIN {X -99.8649,Y 87.4824,Z 169,A 139.6152,B 9.9681,C 0.0739,E1 9.8475,E2 311.3952} C_DIS
LIN {X -102.4956,Y 84.3854,Z 169,A 141.4734,B 9.9681,C 0.076,E1 9.8442,E2 309.5265} C_DIS
LIN {X -105.1854,Y 81.008,Z 169,A 143.0731,B 9.9679,C 0.0851,E1 9.8415,E2 307.9599} C_DIS
LIN {X -108.2901,Y 76.8081,Z 169,A 145.6585,B 9.9679,C 0.0845,E1 9.8372,E2 305.3377} C_DIS
LIN {X -110.9559,Y 72.9034,Z 169,A 147.7304,B 9.9679,C 0.089,E1 9.8339,E2 303.2643} C_DIS
LIN {X -113.4492,Y 68.96,Z 169,A 149.729,B 9.9679,C 0.0943,E1 9.831,E2 301.2695} C_DIS
LIN {X -117.1429,Y 62.4805,Z 169,A 152.8903,B 9.9678,C 0.1036,E1 9.8267,E2 298.1186} C_DIS
LIN {X -118.5955,Y 59.6746,Z 169,A 154.4203,B 9.9678,C 0.1042,E1 9.8247,E2 296.5703} C_DIS
LIN {X -120.1946,Y 56.3858,Z 169,A 155.9409,B 9.9678,C 0.1095,E1 9.8229,E2 295.0583} C_DIS
LIN {X -121.7481,Y 52.9439,Z 169,A 157.5745,B 9.9677,C 0.1138,E1 9.8211,E2 293.4259} C_DIS
LIN {X -123.686,Y 48.2432,Z 169,A 159.6969,B 9.9676,C 0.121,E1 9.8189,E2 291.3144} C_DIS
LIN {X -124.9458,Y 44.8797,Z 169,A 161.379,B 9.9676,C 0.123,E1 9.8172,E2 289.6183} C_DIS
LIN {X -126.3074,Y 40.8941,Z 169,A 163.3042,B 9.9676,C 0.1261,E1 9.8155,E2 287.6823} C_DIS
LIN {X -127.618,Y 36.6033,Z 169,A 165.2367,B 9.9674,C 0.1317,E1 9.814,E2 285.7523} C_DIS
LIN {X -128.455,Y 33.547,Z 169,A 166.6715,B 9.9674,C 0.1343,E1 9.813,E2 284.3109} C_DIS
LIN {X -129.2757,Y 30.231,Z 169,A 168.271,B 9.9674,C 0.1363,E1 9.812,E2 282.698} C_DIS
LIN {X -130.2427,Y 25.7495,Z 169,A 170,B 9.9672,C 0.1464,E1 9.811,E2 281.0009} C_DIS
LIN {X -130.9061,Y 22.1207,Z 169,A 171.4781,B 9.9672,C 0.153,E1 9.8103,E2 279.538} C_DIS
LIN {X -131.2255,Y 20.1387,Z 169,A 173.0228,B 9.9672,C 0.1435,E1 9.8096,E2 277.913} C_DIS
LIN {X -131.8042,Y 15.9175,Z 169,A 174.2613,B 9.967,C 0.1595,E1 9.8092,E2 276.7484} C_DIS
LIN {X -132.1252,Y 12.9891,Z 169,A 175.6992,B 9.967,C 0.1603,E1 9.8088,E2 275.2919} C_DIS
LIN {X -132.3849,Y 10.0024,Z 169,A 176.9094,B 9.967,C 0.1655,E1 9.8085,E2 274.0931} C_DIS
LIN {X -132.5977,Y 6.6014,Z 169,A 178.5205,B 9.967,C 0.1673,E1 9.8083,E2 272.4666} C_DIS
LIN {X -132.7325,Y 2.8757,Z 169,A -179.7541,B 9.9669,C 0.17,E1 9.8081,E2 270.7289} C_DIS
LIN {X -132.7569,Y -1.3307,Z 169,A -177.9359,B 9.9668,C 0.1752,E1 9.8081,E2 268.9121} C_DIS
LIN {X -132.6893,Y -4.4486,Z 169,A -176.7186,B 9.9667,C 0.1814,E1 9.8082,E2 267.7115} C_DIS
LIN {X -132.5593,Y -7.3636,Z 169,A -175.4299,B 9.9667,C 0.1846,E1 9.8084,E2 266.4205} C_DIS
LIN {X -132.3668,Y -10.2509,Z 169,A -173.9398,B 9.9667,C 0.1839,E1 9.8087,E2 264.9026} C_DIS
LIN {X -131.9046,Y -15.0762,Z 169,A -171.9232,B 9.9665,C 0.1913,E1 9.8093,E2 262.8969} C_DIS
LIN {X -131.4735,Y -18.4531,Z 169,A -170.041,B 9.9665,C 0.1882,E1 9.8101,E2 260.9662} C_DIS
LIN {X -130.8259,Y -22.6017,Z 169,A -168.3969,B 9.9664,C 0.1964,E1 9.8108,E2 259.3442} C_DIS
LIN {X -129.8581,Y -27.6168,Z 169,A -166.3786,B 9.9662,C 0.2059,E1 9.8119,E2 257.3502} C_DIS
LIN {X -129.067,Y -31.1023,Z 169,A -164.3315,B 9.9662,C 0.2012,E1 9.8133,E2 255.2433} C_DIS
LIN {X -127.9498,Y -35.4204,Z 169,A -163.1049,B 9.9659,C 0.2191,E1 9.8141,E2 254.1027} C_DIS
LIN {X -126.9765,Y -38.7634,Z 169,A -161.3929,B 9.9659,C 0.2196,E1 9.8155,E2 252.3667} C_DIS
LIN {X -126.0575,Y -41.656,Z 169,A -160.0446,B 9.9659,C 0.2225,E1 9.8167,E2 251.0148} C_DIS
LIN {X -124.595,Y -45.8505,Z 169,A -158.1488,B 9.9657,C 0.2281,E1 9.8184,E2 249.1231} C_DIS
LIN {X -123.3058,Y -49.2086,Z 169,A -156.4616,B 9.9657,C 0.2298,E1 9.8202,E2 247.4207} C_DIS
LIN {X -121.8177,Y -52.7829,Z 169,A -154.9797,B 9.9655,C 0.2376,E1 9.8218,E2 245.9628} C_DIS
LIN {X -120.1054,Y -56.5755,Z 169,A -153.0755,B 9.9655,C 0.2404,E1 9.824,E2 244.0469} C_DIS
LIN {X -118.5507,Y -59.7627,Z 169,A -151.3899,B 9.9655,C 0.2415,E1 9.8261,E2 242.3435} C_DIS
LIN {X -116.7037,Y -63.2966,Z 169,A -149.5918,B 9.9653,C 0.2444,E1 9.8285,E2 240.5372} C_DIS
LIN {X -114.3749,Y -67.4131,Z 169,A -147.686,B 9.9652,C 0.2519,E1 9.8311,E2 238.649} C_DIS
LIN {X -112.7583,Y -70.0834,Z 169,A -146.4163,B 9.965,C 0.2566,E1 9.833,E2 237.3895} C_DIS
LIN {X -111.0559,Y -72.7515,Z 169,A -144.7975,B 9.965,C 0.2552,E1 9.8355,E2 235.7408} C_DIS
LIN {X -109.0744,Y -75.6895,Z 169,A -143.4326,B 9.9649,C 0.2619,E1 9.8376,E2 234.3968} C_DIS
LIN {X -106.9701,Y -78.6352,Z 169,A -141.7738,B 9.9649,C 0.2637,E1 9.8403,E2 232.727} C_DIS
LIN {X -104.8373,Y -81.4571,Z 169,A -140.3951,B 9.9647,C 0.2699,E1 9.8426,E2 231.367} C_DIS
LIN {X -102.9055,Y -83.8844,Z 169,A -138.7927,B 9.9647,C 0.2679,E1 9.8455,E2 229.7333} C_DIS
LIN {X -100.2289,Y -87.0653,Z 169,A -136.9894,B 9.9647,C 0.2716,E1 9.8488,E2 227.9296} C_DIS
LIN {X -97.3849,Y -90.2352,Z 169,A -135.1297,B 9.9645,C 0.275,E1 9.8523,E2 226.068} C_DIS
LIN {X -94.44,Y -93.313,Z 169,A -133.295,B 9.9645,C 0.2788,E1 9.8558,E2 224.2344} C_DIS
LIN {X -91.5226,Y -96.1758,Z 169,A -131.456,B 9.9644,C 0.2808,E1 9.8596,E2 222.387} C_DIS
LIN {X -88.2421,Y -99.1948,Z 169,A -129.5041,B 9.9644,C 0.2838,E1 9.8636,E2 220.4322} C_DIS
LIN {X -84.2087,Y -102.6405,Z 169,A -127.2541,B 9.9642,C 0.2887,E1 9.8684,E2 218.1877} C_DIS
LIN {X -80.9539,Y -105.227,Z 169,A -125.5342,B 9.964,C 0.2932,E1 9.8722,E2 216.4772} C_DIS
LIN {X -78.0218,Y -107.4185,Z 169,A -123.8647,B 9.964,C 0.294,E1 9.8759,E2 214.7971} C_DIS
LIN {X -75.6738,Y -109.0853,Z 169,A -122.4294,B 9.964,C 0.2922,E1 9.8793,E2 213.3384} C_DIS
LIN {X -71.2553,Y -112.022,Z 169,A -120.2717,B 9.9639,C 0.2982,E1 9.8843,E2 211.1973} C_DIS
LIN {X -68.3503,Y -113.8179,Z 169,A -118.7591,B 9.9639,C 0.2996,E1 9.8879,E2 209.6801} C_DIS
LIN {X -63.7367,Y -116.4636,Z 169,A -116.5278,B 9.9637,C 0.3039,E1 9.8933,E2 207.4568} C_DIS
LIN {X -58.0269,Y -119.4109,Z 169,A -113.4073,B 9.9638,C 0.3003,E1 9.9012,E2 204.2936} C_DIS
LIN {X -54.798,Y -120.9263,Z 169,A -112.1009,B 9.9636,C 0.3066,E1 9.9045,E2 203.0159} C_DIS
LIN {X -51.4098,Y -122.4038,Z 169,A -110.6286,B 9.9636,C 0.3108,E1 9.9082,E2 201.5585} C_DIS
LIN {X -48.6532,Y -123.5266,Z 169,A -109.2834,B 9.9636,C 0.3108,E1 9.9117,E2 200.2058} C_DIS
LIN {X -45.8867,Y -124.5815,Z 169,A -107.8936,B 9.9636,C 0.3097,E1 9.9154,E2 198.8021} C_DIS
LIN {X -42.6565,Y -125.7243,Z 169,A -106.5993,B 9.9634,C 0.3147,E1 9.9188,E2 197.5303} C_DIS
LIN {X -39.4914,Y -126.7537,Z 169,A -105.1895,B 9.9634,C 0.3163,E1 9.9225,E2 196.1236} C_DIS
LIN {X -34.6416,Y -128.1631,Z 169,A -102.88,B 9.9634,C 0.3151,E1 9.9288,E2 193.7978} C_DIS
LIN {X -30.8745,Y -129.1219,Z 169,A -101.3275,B 9.9633,C 0.3187,E1 9.9329,E2 192.2601} C_DIS
LIN {X -27.2558,Y -129.936,Z 169,A -99.6032,B 9.9633,C 0.3169,E1 9.9377,E2 190.5204} C_DIS
LIN {X -23.2446,Y -130.711,Z 169,A -97.8579,B 9.9633,C 0.318,E1 9.9425,E2 188.7768} C_DIS
LIN {X -19.2145,Y -131.3647,Z 169,A -96.2709,B 9.9631,C 0.3222,E1 9.9468,E2 187.2106} C_DIS
LIN {X -15.9855,Y -131.7961,Z 169,A -94.6776,B 9.9633,C 0.3186,E1 9.9513,E2 185.5939} C_DIS
LIN {X -11.9819,Y -132.2219,Z 169,A -92.9477,B 9.9633,C 0.3191,E1 9.9561,E2 183.8643} C_DIS
LIN {X -8.9668,Y -132.4605,Z 169,A -91.6691,B 9.9633,C 0.3198,E1 9.9596,E2 182.5885} C_DIS
LIN {X -5.1126,Y -132.6634,Z 169,A -90.0743,B 9.9632,C 0.3213,E1 9.964,E2 181.0016} C_DIS
LIN {X -0.8549,Y -132.7593,Z 169,A -88.2095,B 9.9632,C 0.3206,E1 9.9693,E2 179.1326} C_DIS
LIN {X -0.8549,Y -132.7593,Z 169,A -88.2095,B 9.9632,C 0.3206,E1 9.9693,E2 179.1326} C_DIS
Enddeposition()
LIN {X 0.9667,Y -133.6697,Z 169,A -87.9026,B 9.9615,C 0.3367,E1 9.9687,E2 178.919} C_DIS
Startdeposition()
$VEL.CP = VEL_PRINT
LIN {X -5.9303,Y -133.5446,Z 169,A -91.1024,B 9.9614,C 0.342,E1 9.9597,E2 182.15} C_DIS
LIN {X -9.8352,Y -133.3119,Z 169,A -92.6199,B 9.9614,C 0.3385,E1 9.9555,E2 183.6487} C_DIS
LIN {X -13.5497,Y -132.9878,Z 169,A -94.2877,B 9.9614,C 0.3398,E1 9.9509,E2 185.3257} C_DIS
LIN {X -17.3256,Y -132.5466,Z 169,A -95.8407,B 9.9614,C 0.3378,E1 9.9466,E2 186.8698} C_DIS
LIN {X -20.7245,Y -132.0581,Z 169,A -97.3256,B 9.9614,C 0.3376,E1 9.9425,E2 188.3568} C_DIS
LIN {X -23.9434,Y -131.5128,Z 169,A -98.7746,B 9.9614,C 0.3381,E1 9.9385,E2 189.8123} C_DIS
LIN {X -27.7452,Y -130.7638,Z 169,A -100.4641,B 9.9614,C 0.3379,E1 9.9338,E2 191.5057} C_DIS
LIN {X -31.5741,Y -129.8917,Z 169,A -102.1182,B 9.9615,C 0.3364,E1 9.9293,E2 193.1567} C_DIS
LIN {X -34.7068,Y -129.09,Z 169,A -103.5636,B 9.9615,C 0.3367,E1 9.9254,E2 194.6096} C_DIS
LIN {X -38.7134,Y -127.9459,Z 169,A -105.1068,B 9.9617,C 0.3306,E1 9.9214,E2 196.1235} C_DIS
LIN {X -42.1741,Y -126.8465,Z 169,A -106.7137,B 9.9617,C 0.3304,E1 9.9171,E2 197.7367} C_DIS
LIN {X -44.5998,Y -126.0165,Z 169,A -108.0392,B 9.9617,C 0.334,E1 9.9135,E2 199.0902} C_DIS
LIN {X -49.838,Y -124.0358,Z 169,A -110.0787,B 9.9619,C 0.3246,E1 9.9083,E2 201.0857} C_DIS
LIN {X -53.4186,Y -122.5369,Z 169,A -111.9997,B 9.9619,C 0.328,E1 9.9033,E2 203.0383} C_DIS
LIN {X -56.5925,Y -121.1043,Z 169,A -113.6573,B 9.9618,C 0.3296,E1 9.899,E2 204.7162} C_DIS
LIN {X -62.6845,Y -118.0664,Z 169,A -116.0883,B 9.9622,C 0.3165,E1 9.8931,E2 207.0876} C_DIS
LIN {X -67.2761,Y -115.513,Z 169,A -118.7879,B 9.962,C 0.3223,E1 9.8864,E2 209.8419} C_DIS
LIN {X -71.0043,Y -113.2597,Z 169,A -120.7468,B 9.962,C 0.3214,E1 9.8817,E2 211.8118} C_DIS
LIN {X -74.781,Y -110.8018,Z 169,A -122.629,B 9.9622,C 0.3176,E1 9.8773,E2 213.6876} C_DIS
LIN {X -79.0225,Y -107.8177,Z 169,A -124.6186,B 9.9624,C 0.3095,E1 9.8729,E2 215.6485} C_DIS
LIN {X -81.2448,Y -106.1531,Z 169,A -126.0872,B 9.9623,C 0.3129,E1 9.8695,E2 217.1506} C_DIS
LIN {X -86.8794,Y -101.5939,Z 169,A -129.1292,B 9.9625,C 0.3062,E1 9.863,E2 220.1841} C_DIS
LIN {X -89.8095,Y -99.0124,Z 169,A -130.9198,B 9.9625,C 0.3053,E1 9.8592,E2 221.9884} C_DIS
LIN {X -93.2145,Y -95.8142,Z 169,A -132.951,B 9.9626,C 0.302,E1 9.8551,E2 224.0224} C_DIS
LIN {X -96.2938,Y -92.719,Z 169,A -134.8548,B 9.9627,C 0.2988,E1 9.8514,E2 225.9294} C_DIS
LIN {X -99.2722,Y -89.5231,Z 169,A -136.7282,B 9.9628,C 0.295,E1 9.8479,E2 227.8022} C_DIS
LIN {X -102.0744,Y -86.3141,Z 169,A -138.5488,B 9.963,C 0.2909,E1 9.8445,E2 229.6213} C_DIS
LIN {X -104.8603,Y -82.9077,Z 169,A -140.5212,B 9.963,C 0.2884,E1 9.8411,E2 231.6032} C_DIS
LIN {X -106.6931,Y -80.5343,Z 169,A -141.787,B 9.9631,C 0.2851,E1 9.8389,E2 232.8661} C_DIS
LIN {X -109.4507,Y -76.7455,Z 169,A -143.8423,B 9.9632,C 0.2813,E1 9.8356,E2 234.926} C_DIS
LIN {X -112.9214,Y -71.5401,Z 169,A -146.2044,B 9.9636,C 0.2691,E1 9.832,E2 237.2479} C_DIS
LIN {X -114.5163,Y -68.9584,Z 169,A -147.8433,B 9.9635,C 0.2721,E1 9.8296,E2 238.9269} C_DIS
LIN {X -116.6561,Y -65.2734,Z 169,A -150.0722,B 9.9635,C 0.2749,E1 9.8265,E2 241.203} C_DIS
LIN {X -118.5837,Y -61.6994,Z 169,A -151.3412,B 9.9638,C 0.2619,E1 9.8249,E2 242.4143} C_DIS
LIN {X -120.0135,Y -58.8686,Z 169,A -153.4036,B 9.9635,C 0.2711,E1 9.8223,E2 244.56} C_DIS
LIN {X -122.1894,Y -54.2087,Z 169,A -154.9227,B 9.964,C 0.253,E1 9.8206,E2 245.9956} C_DIS
LIN {X -123.2969,Y -51.6387,Z 169,A -156.184,B 9.964,C 0.251,E1 9.8192,E2 247.2634} C_DIS
LIN {X -124.6854,Y -48.1903,Z 169,A -157.8452,B 9.9641,C 0.2479,E1 9.8175,E2 248.9316} C_DIS
LIN {X -125.8239,Y -45.134,Z 169,A -159.2647,B 9.9641,C 0.2445,E1 9.8161,E2 250.3526} C_DIS
LIN {X -126.9201,Y -41.9531,Z 169,A -160.7203,B 9.9643,C 0.2408,E1 9.8148,E2 251.8087} C_DIS
LIN {X -128.4257,Y -37.0916,Z 169,A -162.8737,B 9.9644,C 0.2343,E1 9.8131,E2 253.9571} C_DIS
LIN {X -130.2456,Y -30.0819,Z 169,A -165.8435,B 9.9647,C 0.2232,E1 9.8111,E2 256.9082} C_DIS
LIN {X -131.5329,Y -23.831,Z 169,A -169.1555,B 9.9647,C 0.2257,E1 9.8092,E2 260.2869} C_DIS
LIN {X -132.0931,Y -20.4979,Z 169,A -170.2194,B 9.9649,C 0.2147,E1 9.8088,E2 261.3035} C_DIS
LIN {X -132.4991,Y -17.6881,Z 169,A -171.5724,B 9.9649,C 0.2136,E1 9.8082,E2 262.6718} C_DIS
LIN {X -132.9728,Y -13.6888,Z 169,A -173.4148,B 9.9649,C 0.2107,E1 9.8077,E2 264.5265} C_DIS
LIN {X -133.326,Y -9.6425,Z 169,A -175.0839,B 9.9651,C 0.2044,E1 9.8073,E2 266.1854} C_DIS
LIN {X -133.5339,Y -6.1503,Z 169,A -176.5653,B 9.9651,C 0.1997,E1 9.8071,E2 267.6633} C_DIS
LIN {X -133.6534,Y -2.3658,Z 169,A -178.2515,B 9.9653,C 0.1961,E1 9.807,E2 269.3554} C_DIS
LIN {X -133.6561,Y 2.2074,Z 169,A 179.7488,B 9.9653,C 0.191,E1 9.807,E2 271.3578} C_DIS
LIN {X -133.5536,Y 5.699,Z 169,A 178.2405,B 9.9654,C 0.1869,E1 9.8072,E2 272.8661} C_DIS
LIN {X -133.3282,Y 9.612,Z 169,A 176.5491,B 9.9655,C 0.1822,E1 9.8075,E2 274.5571} C_DIS
LIN {X -133.0316,Y 13.0949,Z 169,A 175.0787,B 9.9655,C 0.1773,E1 9.8078,E2 276.0227} C_DIS
LIN {X -132.6393,Y 16.6177,Z 169,A 173.3676,B 9.9656,C 0.1763,E1 9.8084,E2 277.7551} C_DIS
LIN {X -131.1413,Y 25.9088,Z 169,A 168.5896,B 9.9656,C 0.1776,E1 9.8108,E2 282.6166} C_DIS
LIN {X -129.8943,Y 31.5636,Z 169,A 166.8247,B 9.9659,C 0.158,E1 9.8118,E2 284.2944} C_DIS
LIN {X -128.3886,Y 37.2182,Z 169,A 164.5309,B 9.9661,C 0.1472,E1 9.8135,E2 286.5601} C_DIS
LIN {X -127.2069,Y 41.0765,Z 169,A 162.5904,B 9.9661,C 0.146,E1 9.8151,E2 288.5239} C_DIS
LIN {X -126.2523,Y 43.9213,Z 169,A 161.2728,B 9.9661,C 0.143,E1 9.8163,E2 289.8437} C_DIS
LIN {X -124.9363,Y 47.5404,Z 169,A 159.4196,B 9.9661,C 0.142,E1 9.8181,E2 291.7192} C_DIS
LIN {X -123.308,Y 51.6122,Z 169,A 157.7397,B 9.9663,C 0.1334,E1 9.8199,E2 293.3734} C_DIS
LIN {X -122.1004,Y 54.4076,Z 169,A 156.3534,B 9.9663,C 0.1313,E1 9.8215,E2 294.7679} C_DIS
LIN {X -120.6347,Y 57.5842,Z 169,A 154.7936,B 9.9663,C 0.1284,E1 9.8233,E2 296.3332} C_DIS
LIN {X -118.7799,Y 61.3235,Z 169,A 153.0431,B 9.9664,C 0.123,E1 9.8255,E2 298.0773} C_DIS
LIN {X -116.9915,Y 64.6699,Z 169,A 150.9844,B 9.9664,C 0.1264,E1 9.8283,E2 300.1852} C_DIS
LIN {X -115.0961,Y 67.9866,Z 169,A 149.021,B 9.9664,C 0.128,E1 9.8312,E2 302.1849} C_DIS
LIN {X -112.2805,Y 72.5422,Z 169,A 146.144,B 9.9663,C 0.1325,E1 9.8357,E2 305.127} C_DIS
LIN {X -107.63,Y 79.2781,Z 169,A 143.9001,B 9.9666,C 0.1017,E1 9.8391,E2 307.2196} C_DIS
LIN {X -105.7623,Y 81.753,Z 169,A 142.4181,B 9.9666,C 0.1013,E1 9.8416,E2 308.7183} C_DIS
LIN {X -102.9989,Y 85.2081,Z 169,A 140.4875,B 9.9666,C 0.0976,E1 9.845,E2 310.651} C_DIS
LIN {X -100.1211,Y 88.5718,Z 169,A 138.5907,B 9.9667,C 0.0934,E1 9.8485,E2 312.5457} C_DIS
LIN {X -96.5574,Y 92.4439,Z 169,A 136.3716,B 9.9667,C 0.0878,E1 9.8527,E2 314.7582} C_DIS
LIN {X -93.8598,Y 95.1823,Z 169,A 134.5891,B 9.9667,C 0.0868,E1 9.8563,E2 316.5549} C_DIS
LIN {X -90.6809,Y 98.2154,Z 169,A 132.7466,B 9.9668,C 0.0823,E1 9.86,E2 318.3907} C_DIS
LIN {X -86.5894,Y 101.8404,Z 169,A 130.5742,B 9.9668,C 0.0745,E1 9.8645,E2 320.5407} C_DIS
LIN {X -84.0507,Y 103.9456,Z 169,A 128.9123,B 9.9668,C 0.0765,E1 9.8682,E2 322.2305} C_DIS
LIN {X -80.8511,Y 106.4534,Z 169,A 126.6059,B 9.9668,C 0.0837,E1 9.8734,E2 324.6012} C_DIS
LIN {X -76.7051,Y 109.4792,Z 169,A 125.2105,B 9.967,C 0.065,E1 9.8764,E2 325.9003} C_DIS
LIN {X -72.491,Y 112.3137,Z 169,A 122.7032,B 9.967,C 0.0676,E1 9.8823,E2 328.4446} C_DIS
LIN {X -68.5592,Y 114.7556,Z 169,A 120.7356,B 9.967,C 0.0642,E1 9.887,E2 330.4084} C_DIS
LIN {X -65.0596,Y 116.7757,Z 169,A 119.1003,B 9.967,C 0.0598,E1 9.8909,E2 332.0309} C_DIS
LIN {X -62.0757,Y 118.3861,Z 169,A 117.6542,B 9.967,C 0.0576,E1 9.8945,E2 333.4748} C_DIS
LIN {X -56.4348,Y 121.1772,Z 169,A 115.1091,B 9.967,C 0.0512,E1 9.9008,E2 335.9997} C_DIS
LIN {X -54.0474,Y 122.2615,Z 169,A 113.8239,B 9.967,C 0.0529,E1 9.9041,E2 337.3031} C_DIS
LIN {X -50.789,Y 123.6518,Z 169,A 112.1157,B 9.967,C 0.0548,E1 9.9086,E2 339.0324} C_DIS
LIN {X -44.9678,Y 125.8838,Z 169,A 109.5899,B 9.967,C 0.0491,E1 9.9152,E2 341.5389} C_DIS
LIN {X -41.8386,Y 126.9583,Z 169,A 107.9105,B 9.967,C 0.0528,E1 9.9197,E2 343.248} C_DIS
LIN {X -34.7287,Y 129.0842,Z 169,A 104.8465,B 9.967,C 0.0479,E1 9.9279,E2 346.296} C_DIS
LIN {X -30.8976,Y 130.0548,Z 169,A 103.2167,B 9.967,C 0.0454,E1 9.9323,E2 347.9171} C_DIS
LIN {X -26.8563,Y 130.9485,Z 169,A 101.3984,B 9.967,C 0.0451,E1 9.9372,E2 349.7394} C_DIS
LIN {X -22.5002,Y 131.7678,Z 169,A 99.486,B 9.967,C 0.0443,E1 9.9425,E2 351.6521} C_DIS
LIN {X -19.0347,Y 132.312,Z 169,A 98.0041,B 9.967,C 0.0432,E1 9.9466,E2 353.1306} C_DIS
LIN {X -15.5229,Y 132.7701,Z 169,A 96.5133,B 9.967,C 0.042,E1 9.9507,E2 354.6174} C_DIS
LIN {X -11.213,Y 133.2031,Z 169,A 94.6325,B 9.967,C 0.042,E1 9.9559,E2 356.4999} C_DIS
LIN {X -6.8029,Y 133.5011,Z 169,A 92.7392,B 9.967,C 0.0415,E1 9.9612,E2 358.3921} C_DIS
LIN {X -3.5338,Y 133.6277,Z 169,A 91.3897,B 9.967,C 0.0403,E1 9.9649,E2 359.7347} C_DIS
LIN {X 0.24,Y 133.675,Z 169,A 89.6832,B 9.967,C 0.042,E1 9.9697,E2 361.451} C_DIS
LIN {X 4.232,Y 133.6083,Z 169,A 88.0853,B 9.967,C 0.0397,E1 9.9742,E2 363.0347} C_DIS
LIN {X 7.8834,Y 133.442,Z 169,A 86.4257,B 9.967,C 0.0418,E1 9.9788,E2 364.7046} C_DIS
LIN {X 11.7949,Y 133.1539,Z 169,A 84.7213,B 9.967,C 0.0427,E1 9.9836,E2 366.4113} C_DIS
LIN {X 15.807,Y 132.7363,Z 169,A 83.012,B 9.967,C 0.0427,E1 9.9883,E2 368.1175} C_DIS
LIN {X 20.2501,Y 132.1315,Z 169,A 81.1118,B 9.967,C 0.043,E1 9.9936,E2 370.0145} C_DIS
LIN {X 23.8065,Y 131.5373,Z 169,A 79.6728,B 9.967,C 0.0415,E1 9.9975,E2 371.4405} C_DIS
LIN {X 26.5657,Y 131.0077,Z 169,A 78.3969,B 9.967,C 0.0436,E1 10.001,E2 372.7246} C_DIS
LIN {X 30.28,Y 130.2003,Z 169,A 76.8207,B 9.967,C 0.0436,E1 10.0053,E2 374.2941} C_DIS
LIN {X 33.9965,Y 129.2794,Z 169,A 74.9869,B 9.967,C 0.0487,E1 10.0103,E2 376.1503} C_DIS
LIN {X 39.0519,Y 127.8423,Z 169,A 72.9896,B 9.967,C 0.045,E1 10.0156,E2 378.117} C_DIS
LIN {X 41.5931,Y 127.04,Z 169,A 71.6964,B 9.967,C 0.0493,E1 10.0191,E2 379.4281} C_DIS
LIN {X 47.2302,Y 125.0525,Z 169,A 69.2375,B 9.967,C 0.0495,E1 10.0255,E2 381.8745} C_DIS
LIN {X 50.7265,Y 123.6776,Z 169,A 67.6391,B 9.967,C 0.0509,E1 10.0296,E2 383.4714} C_DIS
LIN {X 53.1588,Y 122.6492,Z 169,A 66.4605,B 9.967,C 0.0532,E1 10.0327,E2 384.6555} C_DIS
LIN {X 57.2555,Y 120.7917,Z 169,A 64.4414,B 9.967,C 0.0575,E1 10.0378,E2 386.6853} C_DIS
LIN {X 60.0675,Y 119.4193,Z 169,A 63.1719,B 9.967,C 0.0576,E1 10.041,E2 387.9464} C_DIS
LIN {X 63.736,Y 117.5033,Z 169,A 61.4234,B 9.967,C 0.0594,E1 10.0453,E2 389.6921} C_DIS
LIN {X 67.2373,Y 115.5354,Z 169,A 59.6395,B 9.967,C 0.0632,E1 10.0496,E2 391.4834} C_DIS
LIN {X 71.0941,Y 113.203,Z 169,A 57.7439,B 9.967,C 0.0653,E1 10.0541,E2 393.375} C_DIS
LIN {X 77.3093,Y 109.053,Z 169,A 54.6697,B 9.967,C 0.0676,E1 10.0612,E2 396.4344} C_DIS
LIN {X 80.0885,Y 107.0284,Z 169,A 52.8465,B 9.9669,C 0.0779,E1 10.0653,E2 398.2994} C_DIS
LIN {X 83.0347,Y 104.7593,Z 169,A 51.5315,B 9.9669,C 0.0745,E1 10.0682,E2 399.5817} C_DIS
LIN {X 86.5296,Y 101.8912,Z 169,A 49.6435,B 9.9669,C 0.0769,E1 10.0722,E2 401.4643} C_DIS
LIN {X 89.7393,Y 99.0761,Z 169,A 47.824,B 9.9669,C 0.0802,E1 10.076,E2 403.2832} C_DIS
LIN {X 93.0656,Y 95.9583,Z 169,A 45.9133,B 9.9669,C 0.083,E1 10.0798,E2 405.1893} C_DIS
LIN {X 96.1317,Y 92.8865,Z 169,A 44.0585,B 9.9668,C 0.0867,E1 10.0835,E2 407.0441} C_DIS
LIN {X 99.2332,Y 89.5661,Z 169,A 42.126,B 9.9668,C 0.0905,E1 10.0871,E2 408.9757} C_DIS
LIN {X 102.0946,Y 86.2904,Z 169,A 40.257,B 9.9668,C 0.0947,E1 10.0905,E2 410.846} C_DIS
LIN {X 106.9339,Y 80.2152,Z 169,A 37.2397,B 9.9668,C 0.095,E1 10.0957,E2 413.8276} C_DIS
LIN {X 109.9617,Y 76.0118,Z 169,A 35.0495,B 9.9667,C 0.0995,E1 10.0993,E2 416.0154} C_DIS
LIN {X 112.7338,Y 71.8356,Z 169,A 32.7264,B 9.9666,C 0.1088,E1 10.1028,E2 418.3607} C_DIS
LIN {X 114.9261,Y 68.2732,Z 169,A 30.497,B 9.9664,C 0.1234,E1 10.1061,E2 420.6433} C_DIS
LIN {X 117.0841,Y 64.5027,Z 169,A 29.0889,B 9.9664,C 0.1175,E1 10.108,E2 421.9983} C_DIS
LIN {X 118.5263,Y 61.8086,Z 169,A 27.7932,B 9.9664,C 0.1205,E1 10.1096,E2 423.2932} C_DIS
LIN {X 120.4689,Y 57.9312,Z 169,A 25.9998,B 9.9664,C 0.1237,E1 10.1118,E2 425.0799} C_DIS
LIN {X 121.9821,Y 54.6721,Z 169,A 24.4762,B 9.9664,C 0.1274,E1 10.1136,E2 426.6026} C_DIS
LIN {X 123.3647,Y 51.4764,Z 169,A 23.0386,B 9.9664,C 0.1301,E1 10.1152,E2 428.0347} C_DIS
LIN {X 125.1572,Y 46.9506,Z 169,A 20.9228,B 9.9662,C 0.1364,E1 10.1173,E2 430.1555} C_DIS
LIN {X 126.5374,Y 43.0987,Z 169,A 18.9506,B 9.9661,C 0.1464,E1 10.1191,E2 432.1555} C_DIS
LIN {X 127.5616,Y 39.9662,Z 169,A 17.5646,B 9.9661,C 0.1497,E1 10.1203,E2 433.5393} C_DIS
LIN {X 128.4948,Y 36.8557,Z 169,A 16.3112,B 9.9661,C 0.1503,E1 10.1213,E2 434.7773} C_DIS
LIN {X 129.563,Y 32.8962,Z 169,A 14.7544,B 9.9661,C 0.1503,E1 10.1223,E2 436.3113} C_DIS
LIN {X 130.4241,Y 29.3003,Z 169,A 13.0573,B 9.9659,C 0.1576,E1 10.1234,E2 438.0232} C_DIS
LIN {X 131.2783,Y 25.1947,Z 169,A 11.4052,B 9.9659,C 0.1592,E1 10.1243,E2 439.6592} C_DIS
LIN {X 131.8738,Y 21.865,Z 169,A 9.954,B 9.9659,C 0.1634,E1 10.125,E2 441.1119} C_DIS
LIN {X 132.4515,Y 18.0512,Z 169,A 8.2238,B 9.9657,C 0.17,E1 10.1257,E2 442.853} C_DIS
LIN {X 132.9091,Y 14.281,Z 169,A 6.7501,B 9.9657,C 0.171,E1 10.1262,E2 444.3095} C_DIS
LIN {X 133.2754,Y 10.3354,Z 169,A 4.9684,B 9.9656,C 0.178,E1 10.1266,E2 446.1029} C_DIS
LIN {X 133.5105,Y 6.6156,Z 169,A 3.4984,B 9.9656,C 0.1795,E1 10.1268,E2 447.5589} C_DIS
LIN {X 133.6515,Y 2.484,Z 169,A 1.7326,B 9.9655,C 0.1846,E1 10.127,E2 449.3257} C_DIS
LIN {X 133.6645,Y -1.7008,Z 169,A -0.0674,B 9.9654,C 0.19,E1 10.127,E2 451.1282} C_DIS
LIN {X 133.5586,Y -5.5704,Z 169,A -1.6318,B 9.9654,C 0.1925,E1 10.1268,E2 452.6827} C_DIS
LIN {X 133.3287,Y -9.605,Z 169,A -3.3578,B 9.9652,C 0.1974,E1 10.1265,E2 454.4098} C_DIS
LIN {X 132.9733,Y -13.6843,Z 169,A -5.1769,B 9.9651,C 0.2041,E1 10.126,E2 456.2384} C_DIS
LIN {X 132.5153,Y -17.5644,Z 169,A -6.7423,B 9.9651,C 0.2063,E1 10.1255,E2 457.7922} C_DIS
LIN {X 131.8993,Y -21.712,Z 169,A -8.5696,B 9.9649,C 0.2123,E1 10.1247,E2 459.6251} C_DIS
LIN {X 131.2197,Y -25.501,Z 169,A -10.2222,B 9.9649,C 0.2171,E1 10.1238,E2 461.2797} C_DIS
LIN {X 130.3424,Y -29.6581,Z 169,A -11.919,B 9.9648,C 0.2193,E1 10.1228,E2 462.9633} C_DIS
LIN {X 129.4878,Y -33.1924,Z 169,A -13.9772,B 9.9644,C 0.2358,E1 10.1214,E2 465.0838} C_DIS
LIN {X 128.3068,Y -37.4977,Z 169,A -15.4192,B 9.9645,C 0.2299,E1 10.1203,E2 466.4707} C_DIS
LIN {X 126.8837,Y -42.0624,Z 169,A -17.698,B 9.9643,C 0.2411,E1 10.1183,E2 468.7796} C_DIS
LIN {X 125.7415,Y -45.3625,Z 169,A -18.8488,B 9.9643,C 0.237,E1 10.1173,E2 469.8898} C_DIS
LIN {X 124.5043,Y -48.6562,Z 169,A -20.2972,B 9.9643,C 0.2398,E1 10.1158,E2 471.3326} C_DIS
LIN {X 123.1482,Y -51.9949,Z 169,A -21.8547,B 9.9642,C 0.2443,E1 10.1142,E2 472.8934} C_DIS
LIN {X 121.6856,Y -55.3325,Z 169,A -24.2041,B 9.9636,C 0.2673,E1 10.1114,E2 475.3401} C_DIS
LIN {X 119.088,Y -60.7184,Z 169,A -25.5621,B 9.9642,C 0.2454,E1 10.1098,E2 476.5542} C_DIS
LIN {X 114.2267,Y -69.4375,Z 169,A -30.2165,B 9.9637,C 0.2655,E1 10.1034,E2 481.2595} C_DIS
LIN {X 111.925,Y -73.0898,Z 169,A -32.0916,B 9.9635,C 0.2707,E1 10.1006,E2 483.1397} C_DIS
LIN {X 108.691,Y -77.8169,Z 169,A -34.4722,B 9.9635,C 0.275,E1 10.0968,E2 485.5138} C_DIS
LIN {X 105.418,Y -82.1972,Z 169,A -36.6403,B 9.9634,C 0.2765,E1 10.0932,E2 487.6629} C_DIS
LIN {X 103.2924,Y -84.8527,Z 169,A -38.3346,B 9.9631,C 0.2855,E1 10.0901,E2 489.3877} C_DIS
LIN {X 99.9528,Y -88.7622,Z 169,A -40.2018,B 9.9631,C 0.2826,E1 10.0868,E2 491.2159} C_DIS
LIN {X 97.6386,Y -91.3014,Z 169,A -41.8703,B 9.963,C 0.2904,E1 10.0836,E2 492.91} C_DIS
LIN {X 94.6709,Y -94.3751,Z 169,A -43.7541,B 9.9628,C 0.2956,E1 10.0799,E2 494.8021} C_DIS
LIN {X 90.8947,Y -98.0175,Z 169,A -45.7922,B 9.9628,C 0.2954,E1 10.0758,E2 496.8167} C_DIS
LIN {X 88.1371,Y -100.5041,Z 169,A -47.3292,B 9.9628,C 0.2974,E1 10.0726,E2 498.3486} C_DIS
LIN {X 85.4699,Y -102.7821,Z 169,A -48.9811,B 9.9626,C 0.3038,E1 10.069,E2 500.0203} C_DIS
LIN {X 80.1356,Y -106.9935,Z 169,A -51.7257,B 9.9626,C 0.3054,E1 10.063,E2 502.747} C_DIS
LIN {X 75.5064,Y -110.3087,Z 169,A -54.1111,B 9.9624,C 0.3085,E1 10.0576,E2 505.128} C_DIS
LIN {X 72.7063,Y -112.174,Z 169,A -55.709,B 9.9622,C 0.3145,E1 10.0538,E2 506.7464} C_DIS
LIN {X 69.0217,Y -114.4781,Z 169,A -57.8804,B 9.9619,C 0.3246,E1 10.0485,E2 508.9573} C_DIS
LIN {X 65.6627,Y -116.4365,Z 169,A -59.4182,B 9.9619,C 0.3242,E1 10.0448,E2 510.4808} C_DIS
LIN {X 62.737,Y -118.0388,Z 169,A -60.461,B 9.9622,C 0.3176,E1 10.0424,E2 511.4774} C_DIS
LIN {X 59.6508,Y -119.6276,Z 169,A -62.3548,B 9.9618,C 0.3289,E1 10.0375,E2 513.4224} C_DIS
LIN {X 56.4995,Y -121.1472,Z 169,A -63.3388,B 9.9621,C 0.3193,E1 10.0352,E2 514.3443} C_DIS
LIN {X 54.3004,Y -122.1484,Z 169,A -64.5499,B 9.9619,C 0.3246,E1 10.0321,E2 515.5779} C_DIS
LIN {X 51.3268,Y -123.4272,Z 169,A -65.974,B 9.9619,C 0.3272,E1 10.0284,E2 517.0077} C_DIS
LIN {X 47.6614,Y -124.8901,Z 169,A -67.726,B 9.9617,C 0.3305,E1 10.0238,E2 518.7685} C_DIS
LIN {X 44.7999,Y -125.9444,Z 169,A -69.1396,B 9.9617,C 0.3343,E1 10.0201,E2 520.1962} C_DIS
LIN {X 40.013,Y -127.5466,Z 169,A -71.1635,B 9.9617,C 0.3334,E1 10.0147,E2 522.2046} C_DIS
LIN {X 35.3053,Y -128.9282,Z 169,A -73.0629,B 9.9617,C 0.3309,E1 10.0097,E2 524.0805} C_DIS
LIN {X 31.75,Y -129.8493,Z 169,A -74.7714,B 9.9616,C 0.3351,E1 10.005,E2 525.8066} C_DIS
LIN {X 28.1679,Y -130.6725,Z 169,A -76.2411,B 9.9616,C 0.334,E1 10.001,E2 527.2644} C_DIS
LIN {X 24.4091,Y -131.4284,Z 169,A -78.0479,B 9.9615,C 0.3387,E1 9.996,E2 529.0924} C_DIS
LIN {X 20.253,Y -132.131,Z 169,A -79.6527,B 9.9615,C 0.3354,E1 9.9917,E2 530.6735} C_DIS
LIN {X 16.8536,Y -132.6084,Z 169,A -81.3049,B 9.9615,C 0.34,E1 9.987,E2 532.3488} C_DIS
LIN {X 12.782,Y -133.0617,Z 169,A -82.9245,B 9.9615,C 0.3378,E1 9.9826,E2 533.9527} C_DIS
LIN {X 9.349,Y -133.3474,Z 169,A -84.4264,B 9.9615,C 0.3389,E1 9.9784,E2 535.4585} C_DIS
LIN {X 5.2608,Y -133.5707,Z 169,A -86.1463,B 9.9615,C 0.3386,E1 9.9736,E2 537.175} C_DIS
LIN {X 1.4551,Y -133.6684,Z 169,A -87.8773,B 9.9614,C 0.3411,E1 9.9687,E2 538.919} C_DIS
LIN {X 1.4551,Y -133.6684,Z 169,A -87.8773,B 9.9614,C 0.3411,E1 9.9687,E2 538.919} C_DIS
Enddeposition()
LIN {X 0.9743,Y -134.5807,Z 169,A -87.537,B 9.8423,C 0.3392,E1 9.8506,E2 538.5806} C_DIS
Startdeposition()
$VEL.CP = VEL_PRINT
LIN {X 3.87,Y -134.531,Z 169,A -86.0283,B 9.8425,C 0.3331,E1 9.8549,E2 537.0369} C_DIS
LIN {X 7.982,Y -134.35,Z 169,A -84.3095,B 9.8425,C 0.3333,E1 9.8596,E2 535.3215} C_DIS
LIN {X 11.1791,Y -134.1215,Z 169,A -82.9213,B 9.8425,C 0.3324,E1 9.8635,E2 533.9295} C_DIS
LIN {X 14.7583,Y -133.7754,Z 169,A -81.2675,B 9.8426,C 0.329,E1 9.8682,E2 532.2595} C_DIS
LIN {X 18.9735,Y -133.2424,Z 169,A -79.6629,B 9.8426,C 0.3326,E1 9.8725,E2 530.6794} C_DIS
LIN {X 22.0117,Y -132.7743,Z 169,A -78.3088,B 9.8426,C 0.3308,E1 9.8763,E2 529.3187} C_DIS
LIN {X 25.0291,Y -132.2388,Z 169,A -76.9729,B 9.8426,C 0.3293,E1 9.88,E2 527.9781} C_DIS
LIN {X 28.12,Y -131.6162,Z 169,A -75.7988,B 9.8426,C 0.332,E1 9.8831,E2 526.8242} C_DIS
LIN {X 31.1481,Y -130.9329,Z 169,A -74.2608,B 9.8427,C 0.3262,E1 9.8874,E2 525.2581} C_DIS
LIN {X 35.8236,Y -129.7318,Z 169,A -72.2632,B 9.8427,C 0.3257,E1 9.8928,E2 523.2663} C_DIS
LIN {X 39.2895,Y -128.7237,Z 169,A -70.7753,B 9.8427,C 0.3253,E1 9.8967,E2 521.7834} C_DIS
LIN {X 41.903,Y -127.8984,Z 169,A -69.5615,B 9.8428,C 0.3231,E1 9.9,E2 520.5629} C_DIS
LIN {X 45.2138,Y -126.765,Z 169,A -68.0404,B 9.8428,C 0.3207,E1 9.904,E2 519.0366} C_DIS
LIN {X 50.5599,Y -124.7285,Z 169,A -65.6796,B 9.8429,C 0.3196,E1 9.9101,E2 516.6832} C_DIS
LIN {X 54.5428,Y -123.0394,Z 169,A -63.9682,B 9.8429,C 0.3202,E1 9.9145,E2 514.9867} C_DIS
LIN {X 59.1719,Y -120.8812,Z 169,A -61.7155,B 9.8431,C 0.3155,E1 9.9202,E2 512.7225} C_DIS
LIN {X 62.3392,Y -119.2782,Z 169,A -60.2103,B 9.8431,C 0.3134,E1 9.9239,E2 511.2167} C_DIS
LIN {X 65.0601,Y -117.8184,Z 169,A -58.1366,B 9.8437,C 0.2939,E1 9.9292,E2 509.0461} C_DIS
LIN {X 70.0972,Y -114.8931,Z 169,A -56.3215,B 9.8434,C 0.3054,E1 9.9334,E2 507.3128} C_DIS
LIN {X 73.8746,Y -112.5012,Z 169,A -54.4675,B 9.8434,C 0.3033,E1 9.9377,E2 505.4632} C_DIS
LIN {X 79.154,Y -108.8515,Z 169,A -51.806,B 9.8435,C 0.3001,E1 9.9438,E2 502.8081} C_DIS
LIN {X 84.1879,Y -105.0071,Z 169,A -49.0517,B 9.8437,C 0.2937,E1 9.9499,E2 500.044} C_DIS
LIN {X 87.647,Y -102.1372,Z 169,A -47.194,B 9.8437,C 0.2912,E1 9.9538,E2 498.1913} C_DIS
LIN {X 90.9328,Y -99.223,Z 169,A -45.3419,B 9.8439,C 0.2878,E1 9.9577,E2 496.3395} C_DIS
LIN {X 95.1098,Y -95.2271,Z 169,A -42.8957,B 9.844,C 0.283,E1 9.9626,E2 493.8927} C_DIS
LIN {X 98.4244,Y -91.7965,Z 169,A -40.9056,B 9.8441,C 0.2795,E1 9.9664,E2 491.9055} C_DIS
LIN {X 101.4405,Y -88.4521,Z 169,A -38.8376,B 9.8444,C 0.2716,E1 9.9702,E2 489.8167} C_DIS
LIN {X 104.8101,Y -84.4322,Z 169,A -36.8847,B 9.8444,C 0.273,E1 9.9736,E2 487.8965} C_DIS
LIN {X 108.3719,Y -79.8091,Z 169,A -34.6986,B 9.8443,C 0.2743,E1 9.9773,E2 485.7452} C_DIS
LIN {X 110.9741,Y -76.1492,Z 169,A -32.5071,B 9.8446,C 0.2629,E1 9.9809,E2 483.5167} C_DIS
LIN {X 113.2843,Y -72.668,Z 169,A -30.7239,B 9.8447,C 0.2583,E1 9.9836,E2 481.7311} C_DIS
LIN {X 115.3474,Y -69.3473,Z 169,A -28.3086,B 9.8453,C 0.2359,E1 9.9872,E2 479.2194} C_DIS
LIN {X 118.4301,Y -63.9402,Z 169,A -26.3953,B 9.845,C 0.2469,E1 9.9897,E2 477.3962} C_DIS
LIN {X 119.9687,Y -60.9992,Z 169,A -24.1893,B 9.8455,C 0.2239,E1 9.9926,E2 475.0886} C_DIS
LIN {X 122.9092,Y -54.834,Z 169,A -22.2737,B 9.8452,C 0.2402,E1 9.9946,E2 473.2949} C_DIS
LIN {X 124.3461,Y -51.4941,Z 169,A -20.7323,B 9.8452,C 0.2361,E1 9.9963,E2 471.7526} C_DIS
LIN {X 125.7795,Y -47.8903,Z 169,A -19.1674,B 9.8453,C 0.2337,E1 9.9979,E2 470.1967} C_DIS
LIN {X 127.4299,Y -43.3098,Z 169,A -16.9255,B 9.8455,C 0.2238,E1 10,E2 467.9315} C_DIS
LIN {X 128.5189,Y -39.9589,Z 169,A -15.5323,B 9.8455,C 0.2222,E1 10.0011,E2 466.55} C_DIS
LIN {X 130.3094,Y -33.664,Z 169,A -12.8842,B 9.8457,C 0.2176,E1 10.0031,E2 463.9163} C_DIS
LIN {X 131.159,Y -30.1802,Z 169,A -11.3789,B 9.8457,C 0.2138,E1 10.0041,E2 462.4119} C_DIS
LIN {X 131.9343,Y -26.5873,Z 169,A -9.7913,B 9.8459,C 0.2087,E1 10.005,E2 460.8198} C_DIS
LIN {X 132.6856,Y -22.5433,Z 169,A -8.0381,B 9.8459,C 0.2036,E1 10.0058,E2 459.0646} C_DIS
LIN {X 133.2267,Y -19.083,Z 169,A -6.554,B 9.8461,C 0.1994,E1 10.0064,E2 457.5798} C_DIS
LIN {X 133.7452,Y -15.0386,Z 169,A -4.8164,B 9.8461,C 0.1943,E1 10.007,E2 455.8403} C_DIS
LIN {X 134.1106,Y -11.3091,Z 169,A -3.3126,B 9.8462,C 0.1919,E1 10.0074,E2 454.3461} C_DIS
LIN {X 134.3987,Y -7.1187,Z 169,A -1.5298,B 9.8463,C 0.1868,E1 10.0077,E2 452.5623} C_DIS
LIN {X 134.5427,Y -3.4513,Z 169,A 0.0788,B 9.8464,C 0.1811,E1 10.0078,E2 450.9464} C_DIS
LIN {X 134.5874,Y 0.5139,Z 169,A 1.6884,B 9.8464,C 0.1781,E1 10.0078,E2 449.3449} C_DIS
LIN {X 134.5208,Y 4.2369,Z 169,A 3.1975,B 9.8465,C 0.1754,E1 10.0078,E2 447.8437} C_DIS
LIN {X 134.338,Y 8.1771,Z 169,A 4.8348,B 9.8465,C 0.1715,E1 10.0075,E2 446.2099} C_DIS
LIN {X 134.0994,Y 11.4417,Z 169,A 6.2211,B 9.8467,C 0.1676,E1 10.0072,E2 444.8233} C_DIS
LIN {X 133.7234,Y 15.2343,Z 169,A 7.9384,B 9.8467,C 0.1606,E1 10.0067,E2 443.0929} C_DIS
LIN {X 133.2172,Y 19.1496,Z 169,A 9.4672,B 9.8467,C 0.1594,E1 10.0061,E2 441.5812} C_DIS
LIN {X 132.6421,Y 22.804,Z 169,A 11.1043,B 9.8469,C 0.1534,E1 10.0054,E2 439.9351} C_DIS
LIN {X 131.8945,Y 26.7832,Z 169,A 12.691,B 9.8469,C 0.1518,E1 10.0045,E2 438.3637} C_DIS
LIN {X 131.2117,Y 29.9493,Z 169,A 14.1214,B 9.8469,C 0.1467,E1 10.0037,E2 436.9258} C_DIS
LIN {X 130.2093,Y 34.0504,Z 169,A 15.7793,B 9.847,C 0.145,E1 10.0025,E2 435.2836} C_DIS
LIN {X 129.1454,Y 37.8805,Z 169,A 18.1336,B 9.8473,C 0.1243,E1 10.0006,E2 432.846} C_DIS
LIN {X 127.6563,Y 42.6301,Z 169,A 19.6778,B 9.8472,C 0.1323,E1 9.9994,E2 431.3714} C_DIS
LIN {X 126.1076,Y 47.0143,Z 169,A 21.732,B 9.8472,C 0.1251,E1 9.9974,E2 429.3065} C_DIS
LIN {X 124.3426,Y 51.5025,Z 169,A 23.6141,B 9.8472,C 0.1237,E1 9.9954,E2 427.444} C_DIS
LIN {X 122.852,Y 54.9618,Z 169,A 25.0604,B 9.8473,C 0.1232,E1 9.9938,E2 426.0159} C_DIS
LIN {X 121.4643,Y 57.964,Z 169,A 26.5251,B 9.8473,C 0.1182,E1 9.9921,E2 424.5433} C_DIS
LIN {X 120.1511,Y 60.641,Z 169,A 27.8679,B 9.8474,C 0.1132,E1 9.9904,E2 423.1906} C_DIS
LIN {X 118.6727,Y 63.4885,Z 169,A 29.435,B 9.8475,C 0.1049,E1 9.9883,E2 421.598} C_DIS
LIN {X 115.8522,Y 68.5008,Z 169,A 31.7025,B 9.8475,C 0.1031,E1 9.9852,E2 419.3513} C_DIS
LIN {X 113.5107,Y 72.3142,Z 169,A 33.5773,B 9.8475,C 0.0992,E1 9.9824,E2 417.4791} C_DIS
LIN {X 111.0473,Y 76.0425,Z 169,A 35.6586,B 9.8477,C 0.0904,E1 9.9791,E2 415.3748} C_DIS
LIN {X 109.0783,Y 78.841,Z 169,A 36.8565,B 9.8477,C 0.0931,E1 9.9772,E2 414.2079} C_DIS
LIN {X 107.2655,Y 81.2904,Z 169,A 38.5095,B 9.8477,C 0.0818,E1 9.9744,E2 412.5106} C_DIS
LIN {X 104.7439,Y 84.5143,Z 169,A 39.8719,B 9.8477,C 0.0867,E1 9.972,E2 411.1941} C_DIS
LIN {X 101.7706,Y 88.0726,Z 169,A 41.8241,B 9.8477,C 0.0829,E1 9.9685,E2 409.2436} C_DIS
LIN {X 98.9212,Y 91.2612,Z 169,A 43.5645,B 9.8477,C 0.0809,E1 9.9653,E2 407.5123} C_DIS
LIN {X 95.9913,Y 94.3379,Z 169,A 45.4242,B 9.8477,C 0.076,E1 9.9616,E2 405.6457} C_DIS
LIN {X 92.695,Y 97.5794,Z 169,A 47.3924,B 9.8478,C 0.0721,E1 9.9577,E2 403.6768} C_DIS
LIN {X 89.3653,Y 100.6374,Z 169,A 49.2627,B 9.8478,C 0.0696,E1 9.9538,E2 401.8126} C_DIS
LIN {X 86.2534,Y 103.317,Z 169,A 51.0123,B 9.8478,C 0.0664,E1 9.9501,E2 400.0624} C_DIS
LIN {X 83.5671,Y 105.5016,Z 169,A 52.7102,B 9.8478,C 0.0586,E1 9.9463,E2 398.3367} C_DIS
LIN {X 80.7667,Y 107.6607,Z 169,A 53.9797,B 9.8478,C 0.0614,E1 9.9436,E2 397.0958} C_DIS
LIN {X 78.2014,Y 109.5376,Z 169,A 55.786,B 9.8479,C 0.0489,E1 9.9393,E2 395.2337} C_DIS
LIN {X 74.2262,Y 112.2697,Z 169,A 57.3406,B 9.8479,C 0.0569,E1 9.9358,E2 393.7399} C_DIS
LIN {X 70.4848,Y 114.6554,Z 169,A 59.0679,B 9.8479,C 0.0577,E1 9.9318,E2 392.0319} C_DIS
LIN {X 67.3443,Y 116.5277,Z 169,A 60.7305,B 9.8479,C 0.0531,E1 9.9278,E2 390.3564} C_DIS
LIN {X 63.5279,Y 118.6515,Z 169,A 62.647,B 9.8479,C 0.0493,E1 9.923,E2 388.4328} C_DIS
LIN {X 59.9039,Y 120.5201,Z 169,A 64.0596,B 9.8479,C 0.0542,E1 9.9196,E2 387.0593} C_DIS
LIN {X 56.5493,Y 122.1294,Z 169,A 65.8159,B 9.8479,C 0.0485,E1 9.9151,E2 385.2821} C_DIS
LIN {X 53.4877,Y 123.501,Z 169,A 67.1923,B 9.8479,C 0.048,E1 9.9116,E2 383.912} C_DIS
LIN {X 50.7419,Y 124.6551,Z 169,A 68.3754,B 9.8479,C 0.0485,E1 9.9086,E2 382.7393} C_DIS
LIN {X 48.627,Y 125.4945,Z 169,A 69.8549,B 9.8479,C 0.0363,E1 9.9046,E2 381.1979} C_DIS
LIN {X 44.8512,Y 126.8955,Z 169,A 71.3516,B 9.8479,C 0.0395,E1 9.9007,E2 379.728} C_DIS
LIN {X 41.7872,Y 127.937,Z 169,A 72.9661,B 9.848,C 0.0331,E1 9.8964,E2 378.0849} C_DIS
LIN {X 38.053,Y 129.0949,Z 169,A 74.2161,B 9.848,C 0.0408,E1 9.8932,E2 376.8854} C_DIS
LIN {X 33.7763,Y 130.2809,Z 169,A 76.086,B 9.848,C 0.0398,E1 9.8881,E2 375.0183} C_DIS
LIN {X 30.2588,Y 131.141,Z 169,A 77.6237,B 9.848,C 0.0389,E1 9.8839,E2 373.4814} C_DIS
LIN {X 26.5882,Y 131.9341,Z 169,A 79.186,B 9.848,C 0.0388,E1 9.8797,E2 371.9238} C_DIS
LIN {X 22.9605,Y 132.6156,Z 169,A 80.8692,B 9.848,C 0.0357,E1 9.875,E2 370.2276} C_DIS
LIN {X 19.1269,Y 133.2204,Z 169,A 82.4027,B 9.848,C 0.0375,E1 9.8708,E2 368.7089} C_DIS
LIN {X 15.5557,Y 133.6851,Z 169,A 84.0693,B 9.848,C 0.0342,E1 9.8662,E2 367.0268} C_DIS
LIN {X 11.3006,Y 134.1113,Z 169,A 85.753,B 9.848,C 0.0366,E1 9.8615,E2 365.3602} C_DIS
LIN {X 8.0568,Y 134.3454,Z 169,A 87.2157,B 9.848,C 0.0348,E1 9.8574,E2 363.8887} C_DIS
LIN {X 3.7857,Y 134.5334,Z 169,A 88.954,B 9.848,C 0.0364,E1 9.8526,E2 362.1609} C_DIS
LIN {X 0.0157,Y 134.5886,Z 169,A 90.6787,B 9.848,C 0.0339,E1 9.8478,E2 360.4227} C_DIS
LIN {X -3.6823,Y 134.5363,Z 169,A 92.1372,B 9.848,C 0.0365,E1 9.8437,E2 358.9788} C_DIS
LIN {X -7.2064,Y 134.3943,Z 169,A 93.7546,B 9.848,C 0.0343,E1 9.8392,E2 357.3482} C_DIS
LIN {X -11.287,Y 134.1124,Z 169,A 95.4172,B 9.848,C 0.0364,E1 9.8346,E2 355.6959} C_DIS
LIN {X -15.2892,Y 133.7168,Z 169,A 97.0959,B 9.848,C 0.0377,E1 9.8299,E2 354.0223} C_DIS
LIN {X -18.86,Y 133.2586,Z 169,A 98.6186,B 9.848,C 0.0385,E1 9.8257,E2 352.5016} C_DIS
LIN {X -21.6966,Y 132.8269,Z 169,A 99.9288,B 9.848,C 0.0373,E1 9.8221,E2 351.1816} C_DIS
LIN {X -25.0778,Y 132.2295,Z 169,A 101.342,B 9.848,C 0.0391,E1 9.8182,E2 349.775} C_DIS
LIN {X -28.218,Y 131.5951,Z 169,A 102.7187,B 9.848,C 0.0397,E1 9.8144,E2 348.3977} C_DIS
LIN {X -31.6128,Y 130.8209,Z 169,A 104.2949,B 9.848,C 0.0389,E1 9.8101,E2 346.8111} C_DIS
LIN {X -34.6034,Y 130.0618,Z 169,A 106.6495,B 9.848,C 0.0191,E1 9.8035,E2 344.331} C_DIS
LIN {X -42.0156,Y 127.8609,Z 169,A 108.6919,B 9.848,C 0.047,E1 9.7984,E2 342.4428} C_DIS
LIN {X -49.2305,Y 125.2599,Z 169,A 112.1375,B 9.848,C 0.0469,E1 9.7894,E2 338.9783} C_DIS
LIN {X -53.0967,Y 123.67,Z 169,A 113.7739,B 9.848,C 0.0517,E1 9.7852,E2 337.3605} C_DIS
LIN {X -56.2651,Y 122.2608,Z 169,A 115.6818,B 9.848,C 0.0452,E1 9.7802,E2 335.4018} C_DIS
LIN {X -59.2662,Y 120.8347,Z 169,A 117.2025,B 9.848,C 0.045,E1 9.7764,E2 333.8694} C_DIS
LIN {X -62.6481,Y 119.116,Z 169,A 118.3853,B 9.848,C 0.0555,E1 9.7736,E2 332.7402} C_DIS
LIN {X -66.308,Y 117.1212,Z 169,A 120.3448,B 9.848,C 0.0546,E1 9.7687,E2 330.76} C_DIS
LIN {X -69.2675,Y 115.3952,Z 169,A 121.7686,B 9.8479,C 0.0575,E1 9.7653,E2 329.3417} C_DIS
LIN {X -72.8072,Y 113.1952,Z 169,A 123.5643,B 9.8479,C 0.0599,E1 9.7611,E2 327.545} C_DIS
LIN {X -76.4439,Y 110.7719,Z 169,A 125.4691,B 9.8479,C 0.0622,E1 9.7567,E2 325.6366} C_DIS
LIN {X -83.0902,Y 105.8771,Z 169,A 128.9549,B 9.8479,C 0.069,E1 9.7489,E2 322.1576} C_DIS
LIN {X -86.3364,Y 103.2474,Z 169,A 130.5716,B 9.8478,C 0.0753,E1 9.7455,E2 320.5622} C_DIS
LIN {X -88.6981,Y 101.2252,Z 169,A 132.2383,B 9.8478,C 0.0715,E1 9.7419,E2 318.8554} C_DIS
LIN {X -92.5046,Y 97.7593,Z 169,A 134.3369,B 9.8478,C 0.0777,E1 9.7376,E2 316.7703} C_DIS
LIN {X -95.5915,Y 94.743,Z 169,A 136.1817,B 9.8478,C 0.0814,E1 9.7339,E2 314.9264} C_DIS
LIN {X -98.2166,Y 92.0191,Z 169,A 137.9486,B 9.8478,C 0.082,E1 9.7305,E2 313.1422} C_DIS
LIN {X -101.5944,Y 88.2758,Z 169,A 140.0317,B 9.8477,C 0.0879,E1 9.7267,E2 311.069} C_DIS
Enddeposition()
END
